Yaskawa INFORM job: DEMO_ROOF_SIDE_0625_3PAINT_0.JBI

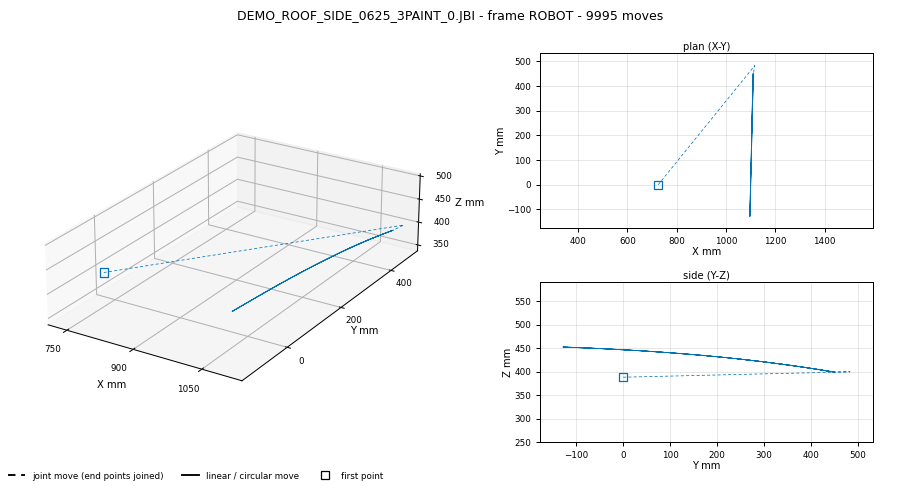
[picture p0: tool path of DEMO_ROOF_SIDE_0625_3PAINT_0.JBI in frame ROBOT, 9995 of 9995 moves have a stored position in this frame; points joined in program order, loops and branches not executed]
/JOB
//NAME DEMO_ROOF_SIDE_0625_3PAINT
//POS
///NPOS 9995,0,0,0,0,0
///TOOL 0
///USER 0
///POSTYPE ROBOT
///RECTAN
///RCONF 1,0,0,0,0,0,0,0,0,0,0,0,0,0,0,0,0,0,0,0,0,0,0,0
C00000=725.000,0.000,388.500,-180.000,-0.000,0.000
///USER 0
///POSTYPE ROBOT
///RECTAN
C00001=1116.924,483.635,399.956,-178.124,16.519,151.125
C00002=1111.077,450.492,399.580,-178.124,16.519,151.125
C00003=1111.072,450.245,399.621,-178.121,16.509,151.122
C00004=1111.067,450.000,399.662,-178.120,16.499,151.119
C00005=1111.061,449.753,399.703,-178.118,16.490,151.116
C00006=1111.056,449.506,399.745,-178.115,16.481,151.114
C00007=1111.050,449.260,399.787,-178.113,16.472,151.111
C00008=1111.045,449.013,399.827,-178.111,16.462,151.108
C00009=1111.039,448.767,399.869,-178.109,16.453,151.105
C00010=1111.034,448.521,399.910,-178.107,16.443,151.102
C00011=1111.028,448.275,399.951,-178.105,16.434,151.099
C00012=1111.023,448.027,399.993,-178.103,16.424,151.096
C00013=1111.017,447.781,400.034,-178.102,16.415,151.094
C00014=1111.012,447.534,400.075,-178.100,16.405,151.091
C00015=1111.007,447.289,400.116,-178.099,16.395,151.088
C00016=1111.002,447.042,400.157,-178.098,16.386,151.085
C00017=1110.996,446.796,400.199,-178.096,16.376,151.082
C00018=1110.991,446.548,400.240,-178.095,16.367,151.080
C00019=1110.985,446.302,400.281,-178.093,16.357,151.077
C00020=1110.980,446.056,400.322,-178.092,16.348,151.074
C00021=1110.975,445.810,400.364,-178.092,16.338,151.072
C00022=1110.969,445.563,400.405,-178.091,16.328,151.069
C00023=1110.963,445.317,400.446,-178.090,16.318,151.066
C00024=1110.957,445.070,400.487,-178.089,16.309,151.064
C00025=1110.952,444.824,400.527,-178.089,16.299,151.061
C00026=1110.947,444.577,400.569,-178.088,16.290,151.058
C00027=1110.941,444.330,400.610,-178.088,16.280,151.056
C00028=1110.935,444.084,400.651,-178.088,16.270,151.053
C00029=1110.930,443.838,400.692,-178.088,16.260,151.051
C00030=1110.925,443.591,400.733,-178.087,16.251,151.048
C00031=1110.919,443.345,400.774,-178.087,16.241,151.046
C00032=1110.915,443.099,400.815,-178.088,16.231,151.043
C00033=1110.909,442.852,400.856,-178.088,16.221,151.041
C00034=1110.903,442.605,400.897,-178.088,16.212,151.038
C00035=1110.898,442.359,400.938,-178.089,16.202,151.036
C00036=1110.892,442.113,400.978,-178.088,16.192,151.033
C00037=1110.887,441.866,401.019,-178.089,16.182,151.031
C00038=1110.881,441.620,401.060,-178.089,16.173,151.028
C00039=1110.876,441.373,401.101,-178.089,16.164,151.026
C00040=1110.870,441.127,401.142,-178.090,16.154,151.024
C00041=1110.864,440.880,401.182,-178.090,16.145,151.021
C00042=1110.859,440.634,401.223,-178.090,16.136,151.019
C00043=1110.853,440.387,401.264,-178.091,16.126,151.017
C00044=1110.848,440.141,401.305,-178.092,16.117,151.014
C00045=1110.843,439.894,401.345,-178.092,16.107,151.012
C00046=1110.837,439.648,401.386,-178.093,16.098,151.010
C00047=1110.831,439.401,401.427,-178.093,16.089,151.007
C00048=1110.826,439.155,401.467,-178.093,16.080,151.005
C00049=1110.820,438.908,401.507,-178.094,16.071,151.003
C00050=1110.814,438.661,401.548,-178.095,16.061,151.001
C00051=1110.809,438.428,401.587,-178.095,16.052,150.998
C00052=1110.804,438.194,401.625,-178.095,16.044,150.996
C00053=1110.799,437.961,401.663,-178.096,16.036,150.994
C00054=1110.794,437.728,401.702,-178.096,16.027,150.992
C00055=1110.788,437.494,401.740,-178.097,16.019,150.990
C00056=1110.783,437.261,401.779,-178.098,16.010,150.988
C00057=1110.778,437.027,401.817,-178.098,16.002,150.986
C00058=1110.773,436.795,401.855,-178.099,15.993,150.984
C00059=1110.767,436.548,401.895,-178.100,15.985,150.982
C00060=1110.761,436.301,401.936,-178.100,15.976,150.980
C00061=1110.756,436.055,401.977,-178.101,15.967,150.978
C00062=1110.751,435.808,402.017,-178.102,15.958,150.976
C00063=1110.745,435.562,402.056,-178.103,15.949,150.973
C00064=1110.740,435.315,402.097,-178.103,15.941,150.971
C00065=1110.734,435.068,402.138,-178.104,15.932,150.969
C00066=1110.729,434.822,402.178,-178.104,15.924,150.967
C00067=1110.723,434.575,402.218,-178.105,15.915,150.965
C00068=1110.718,434.329,402.258,-178.106,15.906,150.963
C00069=1110.712,434.082,402.299,-178.107,15.898,150.961
C00070=1110.707,433.836,402.339,-178.108,15.889,150.959
C00071=1110.701,433.589,402.379,-178.109,15.881,150.957
C00072=1110.696,433.343,402.419,-178.110,15.872,150.955
C00073=1110.690,433.096,402.460,-178.111,15.864,150.953
C00074=1110.684,432.849,402.499,-178.111,15.856,150.951
C00075=1110.679,432.602,402.540,-178.112,15.847,150.949
C00076=1110.674,432.356,402.580,-178.113,15.839,150.947
C00077=1110.668,432.109,402.619,-178.114,15.831,150.945
C00078=1110.662,431.862,402.660,-178.115,15.823,150.943
C00079=1110.657,431.616,402.699,-178.116,15.815,150.942
C00080=1110.651,431.369,402.740,-178.117,15.807,150.940
C00081=1110.646,431.123,402.780,-178.118,15.798,150.938
C00082=1110.640,430.876,402.820,-178.119,15.790,150.936
C00083=1110.635,430.630,402.860,-178.120,15.782,150.934
C00084=1110.629,430.383,402.900,-178.121,15.774,150.932
C00085=1110.623,430.136,402.940,-178.122,15.766,150.930
C00086=1110.618,429.889,402.979,-178.123,15.758,150.928
C00087=1110.612,429.642,403.020,-178.124,15.750,150.927
C00088=1110.607,429.396,403.059,-178.125,15.742,150.925
C00089=1110.602,429.149,403.099,-178.126,15.734,150.923
C00090=1110.596,428.903,403.139,-178.127,15.726,150.921
C00091=1110.590,428.655,403.179,-178.128,15.719,150.919
C00092=1110.585,428.410,403.219,-178.130,15.711,150.918
C00093=1110.579,428.162,403.258,-178.131,15.703,150.916
C00094=1110.574,427.916,403.298,-178.132,15.695,150.914
C00095=1110.567,427.669,403.338,-178.133,15.687,150.912
C00096=1110.563,427.422,403.378,-178.134,15.680,150.911
C00097=1110.557,427.175,403.417,-178.135,15.672,150.909
C00098=1110.551,426.929,403.456,-178.136,15.665,150.907
C00099=1110.546,426.682,403.497,-178.138,15.657,150.906
C00100=1110.540,426.436,403.536,-178.139,15.649,150.904
C00101=1110.534,426.188,403.575,-178.140,15.642,150.902
C00102=1110.529,425.942,403.615,-178.141,15.635,150.901
C00103=1110.523,425.696,403.655,-178.142,15.627,150.899
C00104=1110.518,425.448,403.695,-178.144,15.620,150.897
C00105=1110.513,425.202,403.734,-178.145,15.612,150.896
C00106=1110.507,424.955,403.773,-178.146,15.604,150.894
C00107=1110.502,424.737,403.809,-178.148,15.598,150.893
C00108=1110.497,424.520,403.843,-178.149,15.591,150.891
C00109=1110.492,424.301,403.878,-178.150,15.585,150.890
C00110=1110.487,424.083,403.913,-178.151,15.579,150.888
C00111=1110.483,423.866,403.948,-178.152,15.572,150.887
C00112=1110.477,423.649,403.982,-178.153,15.566,150.885
C00113=1110.472,423.430,404.017,-178.154,15.560,150.884
C00114=1110.468,423.213,404.052,-178.155,15.553,150.883
C00115=1110.462,422.966,404.091,-178.157,15.546,150.881
C00116=1110.456,422.719,404.130,-178.158,15.538,150.880
C00117=1110.451,422.472,404.170,-178.160,15.531,150.878
C00118=1110.446,422.226,404.209,-178.161,15.524,150.877
C00119=1110.440,421.979,404.248,-178.163,15.517,150.875
C00120=1110.434,421.732,404.288,-178.164,15.510,150.874
C00121=1110.429,421.486,404.327,-178.165,15.503,150.872
C00122=1110.422,421.238,404.366,-178.167,15.496,150.871
C00123=1110.417,420.992,404.405,-178.169,15.489,150.869
C00124=1110.412,420.745,404.444,-178.170,15.483,150.868
C00125=1110.407,420.497,404.484,-178.171,15.475,150.866
C00126=1110.401,420.251,404.523,-178.173,15.468,150.865
C00127=1110.395,420.004,404.562,-178.174,15.462,150.863
C00128=1110.389,419.757,404.601,-178.176,15.455,150.862
C00129=1110.384,419.511,404.640,-178.177,15.448,150.860
C00130=1110.378,419.263,404.679,-178.179,15.441,150.859
C00131=1110.373,419.017,404.718,-178.181,15.434,150.858
C00132=1110.367,418.770,404.757,-178.182,15.428,150.856
C00133=1110.361,418.523,404.797,-178.184,15.421,150.855
C00134=1110.356,418.276,404.835,-178.185,15.415,150.854
C00135=1110.351,418.030,404.874,-178.187,15.408,150.852
C00136=1110.345,417.783,404.913,-178.188,15.401,150.851
C00137=1110.339,417.536,404.952,-178.190,15.394,150.850
C00138=1110.334,417.289,404.991,-178.191,15.388,150.848
C00139=1110.328,417.042,405.030,-178.193,15.381,150.847
C00140=1110.323,416.795,405.069,-178.194,15.375,150.845
C00141=1110.317,416.549,405.108,-178.196,15.368,150.844
C00142=1110.311,416.301,405.146,-178.197,15.362,150.843
C00143=1110.306,416.054,405.186,-178.199,15.355,150.842
C00144=1110.301,415.807,405.224,-178.201,15.349,150.840
C00145=1110.295,415.560,405.263,-178.203,15.342,150.839
C00146=1110.288,415.314,405.302,-178.204,15.336,150.838
C00147=1110.283,415.067,405.340,-178.206,15.330,150.836
C00148=1110.277,414.820,405.380,-178.208,15.323,150.835
C00149=1110.272,414.573,405.418,-178.210,15.317,150.834
C00150=1110.267,414.326,405.456,-178.211,15.311,150.833
C00151=1110.261,414.079,405.495,-178.213,15.305,150.832
C00152=1110.255,413.832,405.533,-178.215,15.298,150.830
C00153=1110.249,413.585,405.573,-178.216,15.292,150.829
C00154=1110.244,413.338,405.611,-178.218,15.286,150.828
C00155=1110.238,413.091,405.650,-178.220,15.280,150.827
C00156=1110.232,412.844,405.688,-178.222,15.274,150.826
C00157=1110.227,412.597,405.726,-178.224,15.267,150.824
C00158=1110.222,412.351,405.765,-178.225,15.261,150.823
C00159=1110.216,412.103,405.804,-178.227,15.255,150.822
C00160=1110.211,411.856,405.843,-178.229,15.249,150.821
C00161=1110.205,411.609,405.880,-178.231,15.243,150.820
C00162=1110.199,411.363,405.919,-178.232,15.237,150.818
C00163=1110.194,411.151,405.952,-178.234,15.232,150.818
C00164=1110.190,410.939,405.985,-178.235,15.227,150.817
C00165=1110.185,410.729,406.018,-178.237,15.222,150.816
C00166=1110.180,410.517,406.051,-178.238,15.217,150.815
C00167=1110.176,410.305,406.083,-178.240,15.211,150.814
C00168=1110.171,410.094,406.117,-178.241,15.207,150.813
C00169=1110.166,409.883,406.149,-178.243,15.201,150.812
C00170=1110.161,409.671,406.182,-178.244,15.197,150.811
C00171=1110.156,409.424,406.220,-178.247,15.190,150.810
C00172=1110.150,409.177,406.260,-178.248,15.185,150.809
C00173=1110.144,408.931,406.297,-178.250,15.179,150.808
C00174=1110.139,408.683,406.336,-178.252,15.173,150.806
C00175=1110.134,408.436,406.374,-178.253,15.168,150.805
C00176=1110.128,408.190,406.412,-178.256,15.161,150.804
C00177=1110.123,407.943,406.450,-178.258,15.156,150.803
C00178=1110.116,407.695,406.488,-178.259,15.150,150.802
C00179=1110.111,407.448,406.527,-178.261,15.145,150.801
C00180=1110.105,407.201,406.564,-178.263,15.139,150.800
C00181=1110.100,406.954,406.603,-178.266,15.133,150.799
C00182=1110.095,406.707,406.641,-178.267,15.127,150.798
C00183=1110.089,406.461,406.679,-178.269,15.122,150.797
C00184=1110.084,406.213,406.717,-178.271,15.116,150.796
C00185=1110.077,405.966,406.755,-178.273,15.111,150.795
C00186=1110.072,405.719,406.794,-178.275,15.105,150.794
C00187=1110.066,405.472,406.831,-178.277,15.100,150.793
C00188=1110.061,405.225,406.870,-178.279,15.095,150.792
C00189=1110.055,404.978,406.907,-178.281,15.089,150.791
C00190=1110.049,404.731,406.944,-178.283,15.084,150.791
C00191=1110.044,404.484,406.983,-178.285,15.078,150.790
C00192=1110.038,404.237,407.021,-178.287,15.073,150.789
C00193=1110.033,403.989,407.059,-178.289,15.067,150.788
C00194=1110.027,403.743,407.097,-178.291,15.062,150.787
C00195=1110.021,403.496,407.135,-178.293,15.057,150.786
C00196=1110.016,403.248,407.172,-178.295,15.051,150.785
C00197=1110.010,403.002,407.210,-178.297,15.046,150.784
C00198=1110.004,402.755,407.248,-178.299,15.041,150.783
C00199=1109.999,402.508,407.286,-178.301,15.035,150.782
C00200=1109.993,402.260,407.323,-178.303,15.030,150.781
C00201=1109.987,402.014,407.361,-178.305,15.025,150.781
C00202=1109.982,401.767,407.399,-178.307,15.020,150.780
C00203=1109.977,401.519,407.437,-178.309,15.014,150.779
C00204=1109.971,401.273,407.474,-178.312,15.009,150.778
C00205=1109.966,401.025,407.513,-178.313,15.004,150.777
C00206=1109.960,400.778,407.550,-178.316,14.999,150.776
C00207=1109.954,400.531,407.587,-178.317,14.995,150.775
C00208=1109.949,400.284,407.625,-178.319,14.989,150.775
C00209=1109.943,400.037,407.663,-178.321,14.984,150.774
C00210=1109.937,399.790,407.701,-178.324,14.979,150.773
C00211=1109.932,399.543,407.738,-178.326,14.974,150.772
C00212=1109.926,399.296,407.775,-178.328,14.969,150.771
C00213=1109.921,399.048,407.813,-178.330,14.964,150.771
C00214=1109.915,398.801,407.851,-178.332,14.959,150.770
C00215=1109.909,398.554,407.888,-178.335,14.954,150.769
C00216=1109.904,398.308,407.926,-178.337,14.949,150.768
C00217=1109.898,398.060,407.963,-178.339,14.945,150.767
C00218=1109.892,397.813,408.000,-178.341,14.940,150.767
C00219=1109.888,397.601,408.033,-178.343,14.936,150.766
C00220=1109.883,397.390,408.065,-178.345,14.931,150.765
C00221=1109.878,397.178,408.096,-178.347,14.927,150.765
C00222=1109.873,396.966,408.129,-178.349,14.923,150.764
C00223=1109.868,396.755,408.161,-178.350,14.919,150.763
C00224=1109.863,396.543,408.192,-178.352,14.915,150.763
C00225=1109.858,396.331,408.225,-178.354,14.911,150.762
C00226=1109.854,396.119,408.257,-178.356,14.907,150.762
C00227=1109.848,395.872,408.294,-178.358,14.902,150.761
C00228=1109.842,395.625,408.331,-178.360,14.897,150.760
C00229=1109.837,395.378,408.368,-178.363,14.892,150.760
C00230=1109.831,395.132,408.406,-178.365,14.887,150.759
C00231=1109.826,394.884,408.443,-178.367,14.883,150.758
C00232=1109.820,394.637,408.480,-178.369,14.878,150.757
C00233=1109.815,394.389,408.517,-178.372,14.874,150.757
C00234=1109.809,394.143,408.555,-178.374,14.869,150.756
C00235=1109.803,393.895,408.592,-178.376,14.865,150.755
C00236=1109.797,393.648,408.629,-178.379,14.860,150.755
C00237=1109.792,393.401,408.666,-178.381,14.855,150.754
C00238=1109.787,393.155,408.703,-178.383,14.850,150.753
C00239=1109.781,392.907,408.740,-178.385,14.847,150.753
C00240=1109.775,392.660,408.777,-178.387,14.842,150.752
C00241=1109.770,392.413,408.814,-178.390,14.837,150.752
C00242=1109.764,392.165,408.851,-178.393,14.832,150.751
C00243=1109.758,391.918,408.888,-178.394,14.828,150.750
C00244=1109.752,391.671,408.926,-178.397,14.824,150.750
C00245=1109.746,391.424,408.963,-178.400,14.819,150.749
C00246=1109.741,391.177,408.999,-178.401,14.815,150.749
C00247=1109.736,390.930,409.036,-178.404,14.811,150.748
C00248=1109.729,390.683,409.073,-178.407,14.806,150.748
C00249=1109.724,390.436,409.110,-178.410,14.802,150.747
C00250=1109.718,390.188,409.147,-178.411,14.798,150.746
C00251=1109.713,389.942,409.184,-178.414,14.793,150.746
C00252=1109.707,389.694,409.220,-178.417,14.788,150.745
C00253=1109.701,389.447,409.257,-178.419,14.785,150.745
C00254=1109.696,389.200,409.294,-178.421,14.780,150.744
C00255=1109.690,388.952,409.331,-178.424,14.776,150.744
C00256=1109.684,388.706,409.367,-178.426,14.772,150.743
C00257=1109.679,388.459,409.404,-178.429,14.767,150.743
C00258=1109.673,388.211,409.441,-178.432,14.763,150.742
C00259=1109.667,387.964,409.478,-178.433,14.759,150.741
C00260=1109.662,387.718,409.514,-178.436,14.755,150.741
C00261=1109.656,387.470,409.551,-178.438,14.751,150.740
C00262=1109.650,387.223,409.588,-178.441,14.747,150.740
C00263=1109.645,386.976,409.624,-178.444,14.742,150.739
C00264=1109.640,386.729,409.661,-178.446,14.738,150.739
C00265=1109.633,386.481,409.697,-178.448,14.734,150.738
C00266=1109.628,386.234,409.734,-178.451,14.729,150.738
C00267=1109.623,385.987,409.771,-178.453,14.726,150.738
C00268=1109.617,385.740,409.807,-178.456,14.721,150.737
C00269=1109.611,385.492,409.844,-178.458,14.718,150.737
C00270=1109.606,385.246,409.880,-178.461,14.713,150.736
C00271=1109.600,384.999,409.917,-178.464,14.709,150.736
C00272=1109.594,384.751,409.953,-178.466,14.706,150.735
C00273=1109.589,384.504,409.989,-178.469,14.701,150.735
C00274=1109.583,384.257,410.026,-178.471,14.697,150.734
C00275=1109.573,383.845,410.087,-178.476,14.691,150.734
C00276=1109.564,383.434,410.147,-178.479,14.684,150.733
C00277=1109.555,383.023,410.208,-178.484,14.677,150.732
C00278=1109.546,382.612,410.268,-178.488,14.671,150.732
C00279=1109.540,382.364,410.305,-178.491,14.667,150.731
C00280=1109.534,382.117,410.341,-178.493,14.663,150.731
C00281=1109.529,381.870,410.377,-178.496,14.660,150.730
C00282=1109.523,381.622,410.413,-178.498,14.656,150.730
C00283=1109.517,381.375,410.450,-178.501,14.652,150.730
C00284=1109.512,381.128,410.486,-178.504,14.649,150.729
C00285=1109.506,380.881,410.522,-178.507,14.644,150.729
C00286=1109.500,380.633,410.558,-178.509,14.641,150.728
C00287=1109.495,380.386,410.595,-178.512,14.637,150.728
C00288=1109.489,380.139,410.630,-178.514,14.633,150.728
C00289=1109.483,379.891,410.667,-178.517,14.629,150.728
C00290=1109.478,379.644,410.703,-178.520,14.626,150.727
C00291=1109.472,379.397,410.739,-178.523,14.622,150.727
C00292=1109.467,379.150,410.775,-178.525,14.618,150.726
C00293=1109.461,378.902,410.811,-178.528,14.614,150.726
C00294=1109.455,378.656,410.847,-178.530,14.611,150.726
C00295=1109.450,378.408,410.883,-178.533,14.608,150.726
C00296=1109.444,378.160,410.919,-178.536,14.604,150.725
C00297=1109.438,377.914,410.955,-178.538,14.600,150.725
C00298=1109.433,377.666,410.991,-178.542,14.596,150.725
C00299=1109.427,377.419,411.027,-178.544,14.593,150.724
C00300=1109.421,377.171,411.063,-178.547,14.589,150.724
C00301=1109.416,376.925,411.099,-178.549,14.585,150.724
C00302=1109.410,376.677,411.135,-178.552,14.582,150.723
C00303=1109.405,376.430,411.170,-178.555,14.578,150.723
C00304=1109.399,376.182,411.206,-178.557,14.575,150.723
C00305=1109.393,375.936,411.242,-178.561,14.571,150.723
C00306=1109.388,375.688,411.278,-178.563,14.568,150.722
C00307=1109.382,375.441,411.314,-178.566,14.564,150.722
C00308=1109.376,375.194,411.350,-178.569,14.561,150.722
C00309=1109.371,374.947,411.385,-178.571,14.557,150.722
C00310=1109.366,374.699,411.421,-178.574,14.554,150.721
C00311=1109.360,374.452,411.457,-178.577,14.550,150.721
C00312=1109.354,374.205,411.493,-178.580,14.547,150.721
C00313=1109.348,373.957,411.529,-178.583,14.543,150.721
C00314=1109.342,373.710,411.564,-178.585,14.540,150.720
C00315=1109.336,373.462,411.600,-178.588,14.537,150.720
C00316=1109.331,373.215,411.635,-178.591,14.533,150.720
C00317=1109.325,372.968,411.671,-178.594,14.530,150.720
C00318=1109.319,372.721,411.706,-178.596,14.527,150.719
C00319=1109.314,372.473,411.743,-178.599,14.524,150.719
C00320=1109.309,372.226,411.778,-178.602,14.520,150.719
C00321=1109.303,371.978,411.814,-178.605,14.517,150.719
C00322=1109.297,371.731,411.849,-178.608,14.514,150.719
C00323=1109.291,371.483,411.885,-178.611,14.510,150.719
C00324=1109.286,371.236,411.920,-178.614,14.507,150.718
C00325=1109.280,370.989,411.956,-178.616,14.504,150.718
C00326=1109.274,370.742,411.991,-178.620,14.500,150.718
C00327=1109.266,370.357,412.046,-178.624,14.495,150.718
C00328=1109.256,369.972,412.101,-178.628,14.491,150.718
C00329=1109.248,369.587,412.156,-178.633,14.485,150.717
C00330=1109.240,369.202,412.211,-178.637,14.481,150.717
C00331=1109.233,368.955,412.247,-178.640,14.478,150.717
C00332=1109.228,368.708,412.282,-178.643,14.474,150.717
C00333=1109.222,368.459,412.317,-178.646,14.471,150.717
C00334=1109.217,368.212,412.352,-178.649,14.468,150.717
C00335=1109.211,367.966,412.388,-178.651,14.465,150.716
C00336=1109.206,367.717,412.423,-178.655,14.461,150.716
C00337=1109.200,367.471,412.458,-178.658,14.459,150.716
C00338=1109.194,367.224,412.493,-178.661,14.456,150.716
C00339=1109.188,366.975,412.528,-178.663,14.453,150.716
C00340=1109.183,366.728,412.563,-178.667,14.449,150.716
C00341=1109.177,366.481,412.599,-178.669,14.446,150.716
C00342=1109.172,366.233,412.634,-178.672,14.443,150.716
C00343=1109.166,365.986,412.669,-178.675,14.441,150.716
C00344=1109.160,365.738,412.705,-178.678,14.438,150.716
C00345=1109.155,365.491,412.739,-178.681,14.434,150.715
C00346=1109.149,365.244,412.774,-178.684,14.431,150.715
C00347=1109.143,364.996,412.809,-178.687,14.428,150.715
C00348=1109.138,364.749,412.845,-178.690,14.426,150.715
C00349=1109.132,364.501,412.880,-178.693,14.423,150.715
C00350=1109.126,364.254,412.914,-178.696,14.419,150.715
C00351=1109.121,364.006,412.949,-178.699,14.416,150.715
C00352=1109.115,363.759,412.985,-178.702,14.414,150.715
C00353=1109.110,363.511,413.019,-178.705,14.411,150.715
C00354=1109.104,363.264,413.054,-178.708,14.408,150.715
C00355=1109.098,363.016,413.089,-178.711,14.405,150.715
C00356=1109.092,362.769,413.125,-178.714,14.402,150.715
C00357=1109.087,362.522,413.159,-178.717,14.399,150.715
C00358=1109.081,362.274,413.193,-178.720,14.396,150.715
C00359=1109.075,362.027,413.229,-178.723,14.393,150.715
C00360=1109.070,361.779,413.263,-178.726,14.391,150.715
C00361=1109.064,361.532,413.298,-178.729,14.388,150.715
C00362=1109.058,361.284,413.333,-178.732,14.385,150.715
C00363=1109.053,361.037,413.367,-178.736,14.382,150.715
C00364=1109.047,360.789,413.402,-178.739,14.379,150.715
C00365=1109.041,360.541,413.438,-178.741,14.376,150.715
C00366=1109.036,360.294,413.472,-178.745,14.374,150.715
C00367=1109.030,360.047,413.507,-178.747,14.371,150.715
C00368=1109.024,359.800,413.541,-178.751,14.369,150.715
C00369=1109.019,359.552,413.576,-178.753,14.366,150.715
C00370=1109.013,359.304,413.610,-178.757,14.363,150.715
C00371=1109.008,359.057,413.645,-178.759,14.361,150.715
C00372=1109.002,358.809,413.680,-178.763,14.358,150.715
C00373=1108.996,358.562,413.715,-178.767,14.355,150.715
C00374=1108.991,358.314,413.749,-178.769,14.352,150.715
C00375=1108.985,358.067,413.784,-178.773,14.350,150.715
C00376=1108.980,357.819,413.818,-178.775,14.347,150.715
C00377=1108.973,357.571,413.853,-178.779,14.344,150.715
C00378=1108.968,357.324,413.887,-178.782,14.342,150.715
C00379=1108.959,356.954,413.939,-178.786,14.338,150.715
C00380=1108.950,356.584,413.990,-178.791,14.334,150.715
C00381=1108.942,356.214,414.042,-178.796,14.330,150.715
C00382=1108.934,355.844,414.093,-178.800,14.326,150.715
C00383=1108.928,355.596,414.128,-178.803,14.324,150.716
C00384=1108.922,355.348,414.162,-178.806,14.322,150.716
C00385=1108.917,355.101,414.196,-178.810,14.319,150.716
C00386=1108.911,354.854,414.230,-178.813,14.317,150.716
C00387=1108.906,354.606,414.265,-178.816,14.314,150.716
C00388=1108.900,354.358,414.299,-178.819,14.311,150.716
C00389=1108.894,354.110,414.334,-178.822,14.309,150.716
C00390=1108.889,353.863,414.368,-178.825,14.306,150.716
C00391=1108.883,353.616,414.402,-178.828,14.304,150.716
C00392=1108.878,353.368,414.436,-178.832,14.302,150.716
C00393=1108.872,353.120,414.470,-178.835,14.299,150.716
C00394=1108.866,352.873,414.504,-178.838,14.297,150.717
C00395=1108.860,352.625,414.539,-178.841,14.294,150.717
C00396=1108.855,352.377,414.573,-178.844,14.292,150.717
C00397=1108.849,352.130,414.607,-178.848,14.290,150.717
C00398=1108.843,351.882,414.641,-178.851,14.287,150.717
C00399=1108.838,351.635,414.675,-178.854,14.285,150.717
C00400=1108.832,351.387,414.709,-178.857,14.282,150.717
C00401=1108.826,351.140,414.743,-178.861,14.280,150.718
C00402=1108.820,350.892,414.777,-178.864,14.277,150.718
C00403=1108.815,350.644,414.812,-178.867,14.275,150.718
C00404=1108.809,350.397,414.846,-178.870,14.273,150.718
C00405=1108.804,350.149,414.879,-178.874,14.270,150.718
C00406=1108.798,349.901,414.913,-178.877,14.268,150.718
C00407=1108.792,349.654,414.947,-178.880,14.266,150.719
C00408=1108.787,349.406,414.981,-178.883,14.263,150.719
C00409=1108.781,349.159,415.015,-178.887,14.261,150.719
C00410=1108.775,348.911,415.049,-178.890,14.259,150.719
C00411=1108.770,348.664,415.083,-178.893,14.256,150.719
C00412=1108.763,348.416,415.117,-178.897,14.254,150.719
C00413=1108.758,348.168,415.150,-178.900,14.252,150.720
C00414=1108.753,347.920,415.185,-178.903,14.249,150.720
C00415=1108.747,347.673,415.219,-178.906,14.248,150.720
C00416=1108.741,347.425,415.252,-178.909,14.246,150.720
C00417=1108.735,347.178,415.287,-178.912,14.243,150.720
C00418=1108.730,346.930,415.320,-178.916,14.241,150.720
C00419=1108.724,346.682,415.354,-178.919,14.239,150.721
C00420=1108.718,346.434,415.387,-178.923,14.237,150.721
C00421=1108.713,346.187,415.421,-178.926,14.234,150.721
C00422=1108.707,345.939,415.455,-178.929,14.232,150.721
C00423=1108.701,345.691,415.488,-178.932,14.230,150.721
C00424=1108.696,345.444,415.523,-178.936,14.228,150.722
C00425=1108.691,345.196,415.556,-178.939,14.226,150.722
C00426=1108.685,344.949,415.590,-178.942,14.224,150.722
C00427=1108.679,344.701,415.623,-178.946,14.222,150.722
C00428=1108.673,344.453,415.656,-178.949,14.220,150.723
C00429=1108.667,344.206,415.690,-178.952,14.217,150.723
C00430=1108.662,343.958,415.723,-178.956,14.215,150.723
C00431=1108.654,343.590,415.773,-178.961,14.212,150.724
C00432=1108.645,343.223,415.823,-178.965,14.209,150.724
C00433=1108.636,342.854,415.873,-178.971,14.206,150.724
C00434=1108.628,342.486,415.923,-178.976,14.203,150.725
C00435=1108.622,342.238,415.956,-178.978,14.201,150.725
C00436=1108.616,341.991,415.990,-178.982,14.199,150.725
C00437=1108.611,341.743,416.023,-178.985,14.197,150.725
C00438=1108.605,341.495,416.056,-178.989,14.195,150.726
C00439=1108.600,341.247,416.090,-178.992,14.193,150.726
C00440=1108.594,340.999,416.123,-178.996,14.191,150.726
C00441=1108.589,340.751,416.156,-178.999,14.189,150.727
C00442=1108.583,340.505,416.190,-179.002,14.187,150.727
C00443=1108.577,340.257,416.223,-179.006,14.185,150.727
C00444=1108.571,340.009,416.256,-179.009,14.183,150.727
C00445=1108.566,339.761,416.290,-179.012,14.181,150.728
C00446=1108.560,339.513,416.323,-179.015,14.179,150.728
C00447=1108.555,339.265,416.356,-179.019,14.177,150.728
C00448=1108.549,339.017,416.390,-179.022,14.175,150.728
C00449=1108.543,338.770,416.422,-179.026,14.173,150.729
C00450=1108.537,338.522,416.456,-179.029,14.171,150.729
C00451=1108.532,338.274,416.489,-179.032,14.170,150.729
C00452=1108.527,338.027,416.522,-179.036,14.168,150.730
C00453=1108.521,337.779,416.555,-179.040,14.166,150.730
C00454=1108.515,337.531,416.588,-179.043,14.164,150.730
C00455=1108.509,337.283,416.621,-179.046,14.163,150.731
C00456=1108.503,337.036,416.654,-179.049,14.161,150.731
C00457=1108.498,336.788,416.687,-179.053,14.159,150.731
C00458=1108.492,336.540,416.721,-179.057,14.157,150.732
C00459=1108.486,336.292,416.754,-179.060,14.155,150.732
C00460=1108.481,336.045,416.786,-179.063,14.153,150.732
C00461=1108.476,335.797,416.819,-179.067,14.151,150.733
C00462=1108.469,335.549,416.852,-179.071,14.150,150.733
C00463=1108.464,335.301,416.885,-179.073,14.148,150.733
C00464=1108.458,335.053,416.919,-179.077,14.146,150.734
C00465=1108.452,334.806,416.951,-179.080,14.144,150.734
C00466=1108.447,334.558,416.984,-179.084,14.142,150.734
C00467=1108.441,334.310,417.016,-179.087,14.141,150.735
C00468=1108.435,334.062,417.050,-179.091,14.139,150.735
C00469=1108.430,333.814,417.083,-179.094,14.137,150.736
C00470=1108.423,333.567,417.116,-179.098,14.135,150.736
C00471=1108.419,333.319,417.148,-179.101,14.134,150.736
C00472=1108.413,333.071,417.181,-179.105,14.132,150.737
C00473=1108.407,332.824,417.214,-179.108,14.130,150.737
C00474=1108.402,332.575,417.247,-179.111,14.129,150.737
C00475=1108.395,332.327,417.279,-179.115,14.127,150.738
C00476=1108.391,332.080,417.312,-179.119,14.126,150.738
C00477=1108.385,331.832,417.344,-179.122,14.124,150.738
C00478=1108.378,331.584,417.377,-179.125,14.122,150.739
C00479=1108.373,331.337,417.410,-179.129,14.120,150.739
C00480=1108.367,331.088,417.442,-179.132,14.119,150.740
C00481=1108.361,330.841,417.475,-179.136,14.118,150.740
C00482=1108.356,330.593,417.507,-179.139,14.116,150.740
C00483=1108.347,330.219,417.558,-179.144,14.114,150.741
C00484=1108.338,329.845,417.606,-179.150,14.111,150.742
C00485=1108.329,329.471,417.656,-179.155,14.109,150.742
C00486=1108.321,329.097,417.705,-179.161,14.106,150.743
C00487=1108.315,328.849,417.737,-179.164,14.105,150.743
C00488=1108.309,328.601,417.769,-179.168,14.104,150.744
C00489=1108.304,328.353,417.802,-179.171,14.102,150.744
C00490=1108.298,328.105,417.834,-179.174,14.101,150.745
C00491=1108.292,327.857,417.867,-179.178,14.099,150.745
C00492=1108.286,327.609,417.899,-179.182,14.097,150.746
C00493=1108.281,327.362,417.931,-179.185,14.096,150.746
C00494=1108.275,327.114,417.964,-179.189,14.094,150.746
C00495=1108.269,326.865,417.996,-179.192,14.093,150.747
C00496=1108.264,326.618,418.029,-179.196,14.092,150.747
C00497=1108.258,326.370,418.061,-179.200,14.090,150.748
C00498=1108.252,326.122,418.093,-179.202,14.089,150.748
C00499=1108.246,325.875,418.125,-179.206,14.087,150.749
C00500=1108.241,325.626,418.158,-179.210,14.085,150.749
C00501=1108.235,325.378,418.190,-179.213,14.084,150.750
C00502=1108.229,325.131,418.222,-179.217,14.083,150.750
C00503=1108.223,324.883,418.254,-179.220,14.082,150.751
C00504=1108.218,324.635,418.287,-179.224,14.080,150.751
C00505=1108.213,324.387,418.318,-179.228,14.078,150.751
C00506=1108.206,324.140,418.351,-179.231,14.077,150.752
C00507=1108.200,323.891,418.383,-179.235,14.075,150.752
C00508=1108.195,323.644,418.415,-179.238,14.074,150.753
C00509=1108.189,323.396,418.447,-179.242,14.073,150.753
C00510=1108.184,323.148,418.479,-179.245,14.072,150.754
C00511=1108.178,322.900,418.512,-179.249,14.070,150.754
C00512=1108.172,322.652,418.544,-179.253,14.068,150.755
C00513=1108.167,322.404,418.575,-179.256,14.067,150.755
C00514=1108.161,322.156,418.607,-179.260,14.066,150.756
C00515=1108.155,321.909,418.639,-179.263,14.065,150.756
C00516=1108.150,321.660,418.672,-179.267,14.063,150.757
C00517=1108.145,321.413,418.703,-179.270,14.062,150.757
C00518=1108.139,321.164,418.735,-179.274,14.060,150.758
C00519=1108.133,320.917,418.767,-179.278,14.059,150.758
C00520=1108.127,320.669,418.799,-179.281,14.058,150.759
C00521=1108.122,320.421,418.831,-179.285,14.056,150.759
C00522=1108.116,320.173,418.863,-179.288,14.055,150.759
C00523=1108.111,319.925,418.894,-179.292,14.054,150.760
C00524=1108.105,319.677,418.926,-179.295,14.053,150.760
C00525=1108.099,319.430,418.958,-179.299,14.051,150.761
C00526=1108.093,319.182,418.990,-179.302,14.050,150.762
C00527=1108.088,318.934,419.022,-179.306,14.049,150.762
C00528=1108.082,318.686,419.054,-179.309,14.048,150.763
C00529=1108.077,318.438,419.086,-179.313,14.046,150.763
C00530=1108.071,318.190,419.118,-179.316,14.045,150.764
C00531=1108.066,317.942,419.150,-179.320,14.043,150.764
C00532=1108.060,317.694,419.182,-179.324,14.042,150.765
C00533=1108.055,317.446,419.213,-179.328,14.041,150.765
C00534=1108.049,317.198,419.245,-179.332,14.040,150.766
C00535=1108.040,316.817,419.294,-179.337,14.038,150.766
C00536=1108.031,316.436,419.342,-179.342,14.036,150.767
C00537=1108.023,316.055,419.390,-179.348,14.034,150.768
C00538=1108.014,315.673,419.439,-179.353,14.032,150.769
C00539=1108.009,315.426,419.471,-179.357,14.031,150.769
C00540=1108.003,315.178,419.503,-179.360,14.030,150.770
C00541=1107.997,314.930,419.534,-179.364,14.028,150.770
C00542=1107.992,314.681,419.566,-179.368,14.028,150.771
C00543=1107.985,314.434,419.597,-179.372,14.026,150.772
C00544=1107.980,314.187,419.628,-179.375,14.025,150.772
C00545=1107.974,313.938,419.660,-179.378,14.025,150.773
C00546=1107.968,313.690,419.691,-179.383,14.023,150.773
C00547=1107.962,313.442,419.723,-179.386,14.022,150.774
C00548=1107.957,313.194,419.754,-179.390,14.021,150.774
C00549=1107.951,312.946,419.786,-179.393,14.020,150.775
C00550=1107.945,312.699,419.817,-179.397,14.019,150.776
C00551=1107.939,312.450,419.848,-179.401,14.018,150.776
C00552=1107.934,312.202,419.880,-179.405,14.017,150.777
C00553=1107.928,311.955,419.910,-179.408,14.016,150.777
C00554=1107.922,311.706,419.942,-179.412,14.014,150.778
C00555=1107.917,311.459,419.974,-179.416,14.014,150.779
C00556=1107.911,311.211,420.004,-179.419,14.013,150.779
C00557=1107.905,310.963,420.036,-179.423,14.012,150.780
C00558=1107.900,310.715,420.067,-179.427,14.011,150.780
C00559=1107.893,310.467,420.098,-179.430,14.009,150.781
C00560=1107.888,310.219,420.129,-179.434,14.009,150.782
C00561=1107.882,309.971,420.160,-179.438,14.007,150.782
C00562=1107.876,309.723,420.192,-179.441,14.007,150.783
C00563=1107.871,309.475,420.223,-179.446,14.005,150.783
C00564=1107.865,309.227,420.254,-179.449,14.004,150.784
C00565=1107.859,308.978,420.285,-179.452,14.004,150.785
C00566=1107.853,308.731,420.316,-179.456,14.003,150.785
C00567=1107.848,308.483,420.347,-179.460,14.002,150.786
C00568=1107.842,308.236,420.378,-179.464,14.000,150.786
C00569=1107.836,307.987,420.409,-179.467,14.000,150.787
C00570=1107.831,307.739,420.440,-179.472,13.999,150.788
C00571=1107.825,307.492,420.472,-179.475,13.998,150.788
C00572=1107.820,307.243,420.503,-179.478,13.997,150.789
C00573=1107.814,306.995,420.533,-179.483,13.996,150.789
C00574=1107.808,306.748,420.565,-179.486,13.995,150.790
C00575=1107.803,306.500,420.595,-179.490,13.994,150.791
C00576=1107.797,306.251,420.626,-179.493,13.993,150.791
C00577=1107.791,306.003,420.657,-179.498,13.992,150.792
C00578=1107.786,305.756,420.689,-179.501,13.991,150.792
C00579=1107.780,305.508,420.719,-179.504,13.990,150.793
C00580=1107.775,305.260,420.750,-179.509,13.989,150.794
C00581=1107.768,305.011,420.781,-179.512,13.989,150.794
C00582=1107.763,304.763,420.811,-179.516,13.987,150.795
C00583=1107.757,304.516,420.843,-179.519,13.986,150.796
C00584=1107.751,304.268,420.873,-179.523,13.986,150.796
C00585=1107.746,304.020,420.904,-179.527,13.985,150.797
C00586=1107.740,303.772,420.934,-179.531,13.984,150.798
C00587=1107.732,303.394,420.981,-179.536,13.983,150.799
C00588=1107.723,303.014,421.028,-179.543,13.981,150.800
C00589=1107.714,302.636,421.075,-179.548,13.979,150.800
C00590=1107.705,302.257,421.122,-179.554,13.978,150.801
C00591=1107.700,302.009,421.153,-179.557,13.978,150.802
C00592=1107.694,301.762,421.183,-179.561,13.976,150.803
C00593=1107.689,301.513,421.214,-179.565,13.976,150.803
C00594=1107.683,301.266,421.245,-179.568,13.975,150.804
C00595=1107.678,301.018,421.275,-179.573,13.974,150.805
C00596=1107.673,300.770,421.306,-179.576,13.974,150.806
C00597=1107.667,300.521,421.336,-179.580,13.972,150.806
C00598=1107.661,300.273,421.366,-179.584,13.972,150.807
C00599=1107.655,300.025,421.397,-179.587,13.971,150.807
C00600=1107.650,299.777,421.428,-179.591,13.970,150.808
C00601=1107.644,299.529,421.458,-179.595,13.969,150.809
C00602=1107.639,299.281,421.489,-179.598,13.969,150.809
C00603=1107.633,299.033,421.519,-179.603,13.967,150.810
C00604=1107.627,298.785,421.550,-179.606,13.967,150.811
C00605=1107.621,298.537,421.580,-179.610,13.966,150.811
C00606=1107.617,298.289,421.610,-179.614,13.965,150.812
C00607=1107.611,298.041,421.641,-179.617,13.964,150.813
C00608=1107.605,297.793,421.671,-179.621,13.964,150.813
C00609=1107.599,297.545,421.701,-179.625,13.963,150.814
C00610=1107.593,297.297,421.732,-179.629,13.963,150.815
C00611=1107.588,297.049,421.761,-179.632,13.962,150.816
C00612=1107.583,296.801,421.792,-179.637,13.961,150.816
C00613=1107.577,296.553,421.823,-179.640,13.960,150.817
C00614=1107.571,296.305,421.853,-179.644,13.960,150.818
C00615=1107.565,296.056,421.883,-179.648,13.959,150.818
C00616=1107.559,295.808,421.913,-179.652,13.958,150.819
C00617=1107.553,295.560,421.944,-179.655,13.958,150.820
C00618=1107.548,295.312,421.973,-179.660,13.957,150.820
C00619=1107.542,295.064,422.004,-179.663,13.956,150.821
C00620=1107.536,294.816,422.034,-179.667,13.956,150.822
C00621=1107.531,294.568,422.064,-179.670,13.955,150.823
C00622=1107.525,294.320,422.094,-179.675,13.954,150.823
C00623=1107.519,294.072,422.124,-179.678,13.954,150.824
C00624=1107.514,293.824,422.154,-179.682,13.953,150.825
C00625=1107.508,293.576,422.184,-179.686,13.952,150.825
C00626=1107.502,293.327,422.214,-179.690,13.951,150.826
C00627=1107.496,293.080,422.244,-179.693,13.951,150.827
C00628=1107.491,292.831,422.274,-179.698,13.950,150.828
C00629=1107.485,292.583,422.304,-179.701,13.949,150.828
C00630=1107.479,292.335,422.335,-179.705,13.949,150.829
C00631=1107.474,292.087,422.364,-179.709,13.949,150.830
C00632=1107.468,291.839,422.394,-179.713,13.948,150.830
C00633=1107.462,291.591,422.424,-179.716,13.947,150.831
C00634=1107.457,291.342,422.454,-179.720,13.947,150.832
C00635=1107.451,291.094,422.484,-179.724,13.946,150.833
C00636=1107.446,290.846,422.514,-179.728,13.945,150.833
C00637=1107.440,290.598,422.544,-179.732,13.945,150.834
C00638=1107.435,290.350,422.574,-179.735,13.945,150.835
C00639=1107.426,289.985,422.617,-179.741,13.943,150.836
C00640=1107.418,289.621,422.661,-179.747,13.943,150.837
C00641=1107.410,289.256,422.705,-179.753,13.942,150.838
C00642=1107.401,288.891,422.749,-179.758,13.941,150.839
C00643=1107.395,288.643,422.779,-179.762,13.940,150.840
C00644=1107.389,288.395,422.808,-179.766,13.940,150.841
C00645=1107.384,288.147,422.838,-179.769,13.940,150.842
C00646=1107.378,287.899,422.868,-179.773,13.939,150.842
C00647=1107.372,287.651,422.898,-179.778,13.938,150.843
C00648=1107.367,287.403,422.926,-179.781,13.938,150.844
C00649=1107.361,287.155,422.956,-179.785,13.938,150.845
C00650=1107.355,286.907,422.986,-179.789,13.937,150.845
C00651=1107.350,286.658,423.016,-179.792,13.937,150.846
C00652=1107.343,286.410,423.045,-179.797,13.936,150.847
C00653=1107.338,286.162,423.075,-179.800,13.936,150.848
C00654=1107.332,285.913,423.104,-179.804,13.935,150.848
C00655=1107.327,285.665,423.134,-179.808,13.935,150.849
C00656=1107.321,285.418,423.163,-179.812,13.934,150.850
C00657=1107.315,285.170,423.193,-179.816,13.934,150.851
C00658=1107.310,284.921,423.223,-179.820,13.933,150.851
C00659=1107.304,284.673,423.252,-179.823,13.933,150.852
C00660=1107.298,284.425,423.281,-179.827,13.933,150.853
C00661=1107.293,284.176,423.311,-179.832,13.932,150.854
C00662=1107.287,283.929,423.340,-179.835,13.931,150.855
C00663=1107.282,283.680,423.369,-179.839,13.931,150.855
C00664=1107.276,283.432,423.399,-179.843,13.931,150.856
C00665=1107.270,283.184,423.428,-179.847,13.930,150.857
C00666=1107.264,282.935,423.457,-179.851,13.930,150.858
C00667=1107.259,282.688,423.487,-179.854,13.929,150.858
C00668=1107.253,282.440,423.516,-179.858,13.929,150.859
C00669=1107.248,282.191,423.545,-179.862,13.929,150.860
C00670=1107.242,281.943,423.575,-179.866,13.928,150.861
C00671=1107.236,281.695,423.604,-179.870,13.927,150.862
C00672=1107.231,281.447,423.633,-179.874,13.927,150.862
C00673=1107.225,281.199,423.662,-179.878,13.927,150.863
C00674=1107.219,280.950,423.692,-179.881,13.926,150.864
C00675=1107.213,280.702,423.721,-179.885,13.926,150.865
C00676=1107.208,280.454,423.750,-179.890,13.926,150.866
C00677=1107.202,280.206,423.779,-179.893,13.925,150.866
C00678=1107.197,279.957,423.808,-179.897,13.925,150.867
C00679=1107.190,279.709,423.837,-179.901,13.925,150.868
C00680=1107.185,279.461,423.867,-179.904,13.924,150.869
C00681=1107.179,279.213,423.896,-179.909,13.924,150.870
C00682=1107.174,278.965,423.925,-179.913,13.923,150.870
C00683=1107.168,278.716,423.954,-179.916,13.923,150.871
C00684=1107.162,278.468,423.983,-179.920,13.923,150.872
C00685=1107.157,278.220,424.012,-179.924,13.923,150.873
C00686=1107.151,277.972,424.042,-179.928,13.923,150.874
C00687=1107.145,277.723,424.070,-179.932,13.921,150.874
C00688=1107.139,277.475,424.099,-179.936,13.921,150.875
C00689=1107.134,277.227,424.128,-179.940,13.921,150.876
C00690=1107.128,276.978,424.157,-179.944,13.921,150.877
C00691=1107.120,276.623,424.199,-179.950,13.920,150.878
C00692=1107.112,276.269,424.240,-179.955,13.920,150.879
C00693=1107.104,275.913,424.281,-179.961,13.919,150.880
C00694=1107.096,275.558,424.322,-179.966,13.919,150.882
C00695=1107.090,275.309,424.352,-179.970,13.919,150.883
C00696=1107.085,275.061,424.380,-179.974,13.919,150.883
C00697=1107.079,274.813,424.409,-179.977,13.919,150.884
C00698=1107.073,274.564,424.438,-179.982,13.918,150.885
C00699=1107.068,274.317,424.466,-179.986,13.918,150.886
C00700=1107.061,274.069,424.495,-179.990,13.918,150.887
C00701=1107.056,273.820,424.524,-179.993,13.917,150.887
C00702=1107.051,273.572,424.553,-179.997,13.917,150.888
C00703=1107.045,273.323,424.581,179.999,13.917,150.889
C00704=1107.038,273.075,424.610,179.995,13.917,150.890
C00705=1107.033,272.827,424.638,179.990,13.916,150.891
C00706=1107.028,272.578,424.667,179.987,13.916,150.892
C00707=1107.022,272.330,424.696,179.983,13.916,150.893
C00708=1107.016,272.082,424.724,179.979,13.915,150.893
C00709=1107.010,271.834,424.753,179.975,13.915,150.894
C00710=1107.005,271.585,424.782,179.971,13.915,150.895
C00711=1106.999,271.337,424.811,179.968,13.915,150.896
C00712=1106.993,271.089,424.839,179.964,13.915,150.897
C00713=1106.988,270.841,424.867,179.959,13.914,150.898
C00714=1106.982,270.592,424.896,179.955,13.914,150.898
C00715=1106.976,270.344,424.924,179.951,13.914,150.899
C00716=1106.971,270.095,424.953,179.947,13.914,150.900
C00717=1106.965,269.847,424.982,179.944,13.914,150.901
C00718=1106.959,269.599,425.010,179.940,13.914,150.902
C00719=1106.954,269.350,425.038,179.936,13.913,150.903
C00720=1106.948,269.102,425.066,179.932,13.913,150.903
C00721=1106.942,268.854,425.095,179.928,13.913,150.904
C00722=1106.937,268.606,425.123,179.925,13.913,150.905
C00723=1106.931,268.357,425.152,179.920,13.912,150.906
C00724=1106.925,268.109,425.180,179.916,13.912,150.907
C00725=1106.919,267.861,425.209,179.912,13.912,150.908
C00726=1106.913,267.612,425.237,179.908,13.912,150.909
C00727=1106.908,267.364,425.265,179.904,13.912,150.909
C00728=1106.902,267.116,425.293,179.901,13.912,150.910
C00729=1106.897,266.867,425.322,179.897,13.912,150.911
C00730=1106.891,266.618,425.350,179.893,13.912,150.912
C00731=1106.886,266.371,425.379,179.889,13.912,150.913
C00732=1106.880,266.122,425.407,179.885,13.912,150.914
C00733=1106.874,265.874,425.435,179.881,13.912,150.915
C00734=1106.868,265.626,425.463,179.877,13.912,150.916
C00735=1106.863,265.377,425.491,179.873,13.911,150.916
C00736=1106.857,265.129,425.520,179.869,13.911,150.917
C00737=1106.852,264.881,425.548,179.865,13.911,150.918
C00738=1106.846,264.632,425.576,179.861,13.911,150.919
C00739=1106.840,264.384,425.603,179.857,13.911,150.920
C00740=1106.834,264.135,425.632,179.853,13.911,150.921
C00741=1106.828,263.887,425.659,179.849,13.911,150.922
C00742=1106.823,263.639,425.688,179.845,13.911,150.923
C00743=1106.815,263.286,425.728,179.840,13.911,150.924
C00744=1106.807,262.934,425.767,179.834,13.910,150.925
C00745=1106.798,262.583,425.807,179.828,13.911,150.927
C00746=1106.790,262.229,425.846,179.823,13.911,150.928
C00747=1106.784,261.981,425.874,179.819,13.911,150.929
C00748=1106.779,261.733,425.902,179.815,13.911,150.930
C00749=1106.772,261.485,425.930,179.811,13.911,150.931
C00750=1106.767,261.237,425.958,179.807,13.911,150.931
C00751=1106.761,260.988,425.986,179.802,13.910,150.932
C00752=1106.756,260.740,426.014,179.799,13.910,150.933
C00753=1106.749,260.491,426.041,179.794,13.910,150.934
C00754=1106.744,260.243,426.069,179.791,13.910,150.935
C00755=1106.738,259.994,426.097,179.787,13.910,150.936
C00756=1106.733,259.746,426.125,179.783,13.910,150.937
C00757=1106.727,259.498,426.153,179.779,13.910,150.938
C00758=1106.721,259.249,426.180,179.775,13.910,150.939
C00759=1106.716,259.001,426.208,179.771,13.910,150.940
C00760=1106.710,258.752,426.237,179.767,13.910,150.940
C00761=1106.704,258.504,426.264,179.763,13.910,150.941
C00762=1106.699,258.255,426.291,179.759,13.910,150.942
C00763=1106.693,258.007,426.320,179.755,13.910,150.943
C00764=1106.687,257.759,426.347,179.751,13.910,150.944
C00765=1106.681,257.510,426.375,179.747,13.910,150.945
C00766=1106.676,257.262,426.403,179.743,13.910,150.946
C00767=1106.669,257.014,426.430,179.739,13.910,150.947
C00768=1106.664,256.764,426.457,179.735,13.911,150.948
C00769=1106.659,256.516,426.485,179.731,13.911,150.949
C00770=1106.653,256.268,426.512,179.727,13.910,150.950
C00771=1106.647,256.019,426.540,179.723,13.910,150.950
C00772=1106.641,255.772,426.568,179.720,13.910,150.951
C00773=1106.636,255.523,426.595,179.715,13.911,150.952
C00774=1106.630,255.274,426.623,179.711,13.911,150.953
C00775=1106.624,255.026,426.650,179.708,13.911,150.954
C00776=1106.619,254.778,426.678,179.704,13.911,150.955
C00777=1106.613,254.529,426.705,179.699,13.911,150.956
C00778=1106.607,254.281,426.733,179.696,13.911,150.957
C00779=1106.602,254.032,426.760,179.692,13.911,150.958
C00780=1106.596,253.784,426.788,179.688,13.911,150.959
C00781=1106.590,253.535,426.815,179.684,13.911,150.960
C00782=1106.584,253.287,426.842,179.680,13.911,150.961
C00783=1106.579,253.038,426.870,179.676,13.911,150.961
C00784=1106.573,252.790,426.896,179.672,13.911,150.962
C00785=1106.567,252.541,426.925,179.668,13.911,150.963
C00786=1106.562,252.293,426.951,179.664,13.911,150.964
C00787=1106.556,252.045,426.979,179.660,13.911,150.965
C00788=1106.550,251.797,427.006,179.656,13.911,150.966
C00789=1106.545,251.548,427.033,179.652,13.912,150.967
C00790=1106.539,251.299,427.061,179.648,13.912,150.968
C00791=1106.534,251.051,427.088,179.644,13.912,150.969
C00792=1106.528,250.802,427.115,179.640,13.912,150.970
C00793=1106.523,250.554,427.142,179.636,13.912,150.971
C00794=1106.516,250.305,427.170,179.632,13.912,150.972
C00795=1106.509,249.950,427.208,179.626,13.912,150.973
C00796=1106.501,249.595,427.248,179.620,13.912,150.974
C00797=1106.493,249.240,427.286,179.615,13.912,150.976
C00798=1106.485,248.885,427.324,179.609,13.912,150.977
C00799=1106.479,248.637,427.352,179.605,13.913,150.978
C00800=1106.473,248.388,427.379,179.601,13.913,150.979
C00801=1106.468,248.139,427.406,179.597,13.913,150.980
C00802=1106.462,247.891,427.433,179.594,13.913,150.981
C00803=1106.457,247.643,427.460,179.589,13.913,150.982
C00804=1106.452,247.394,427.487,179.585,13.913,150.983
C00805=1106.445,247.146,427.514,179.582,13.913,150.983
C00806=1106.439,246.897,427.541,179.577,13.913,150.984
C00807=1106.434,246.649,427.568,179.573,13.913,150.985
C00808=1106.428,246.400,427.595,179.569,13.914,150.986
C00809=1106.423,246.152,427.622,179.565,13.914,150.987
C00810=1106.417,245.903,427.649,179.561,13.914,150.988
C00811=1106.412,245.655,427.676,179.557,13.914,150.989
C00812=1106.406,245.407,427.702,179.553,13.914,150.990
C00813=1106.400,245.158,427.729,179.549,13.914,150.991
C00814=1106.395,244.909,427.757,179.546,13.915,150.992
C00815=1106.389,244.660,427.783,179.542,13.915,150.993
C00816=1106.383,244.412,427.810,179.538,13.915,150.994
C00817=1106.377,244.164,427.837,179.534,13.915,150.995
C00818=1106.372,243.915,427.864,179.530,13.915,150.996
C00819=1106.366,243.667,427.890,179.526,13.916,150.997
C00820=1106.361,243.418,427.917,179.522,13.916,150.998
C00821=1106.355,243.170,427.944,179.518,13.916,150.999
C00822=1106.349,242.922,427.970,179.514,13.916,151.000
C00823=1106.344,242.673,427.998,179.510,13.916,151.001
C00824=1106.339,242.424,428.024,179.506,13.916,151.002
C00825=1106.333,242.176,428.050,179.501,13.917,151.003
C00826=1106.326,241.927,428.077,179.498,13.917,151.003
C00827=1106.321,241.678,428.104,179.494,13.917,151.004
C00828=1106.315,241.430,428.130,179.489,13.917,151.005
C00829=1106.309,241.181,428.157,179.485,13.917,151.006
C00830=1106.304,240.932,428.183,179.482,13.918,151.007
C00831=1106.298,240.684,428.210,179.478,13.918,151.008
C00832=1106.292,240.436,428.236,179.474,13.919,151.009
C00833=1106.286,240.187,428.263,179.470,13.919,151.010
C00834=1106.281,239.939,428.290,179.466,13.919,151.011
C00835=1106.275,239.690,428.316,179.462,13.919,151.012
C00836=1106.269,239.442,428.342,179.458,13.919,151.013
C00837=1106.264,239.193,428.369,179.454,13.919,151.014
C00838=1106.258,238.944,428.395,179.449,13.920,151.015
C00839=1106.252,238.696,428.421,179.446,13.920,151.016
C00840=1106.247,238.448,428.448,179.441,13.920,151.017
C00841=1106.241,238.199,428.474,179.438,13.921,151.018
C00842=1106.235,237.950,428.501,179.434,13.921,151.019
C00843=1106.229,237.702,428.527,179.430,13.921,151.020
C00844=1106.224,237.453,428.553,179.426,13.922,151.021
C00845=1106.218,237.205,428.580,179.422,13.922,151.022
C00846=1106.212,236.956,428.607,179.418,13.922,151.023
C00847=1106.205,236.595,428.645,179.412,13.923,151.024
C00848=1106.196,236.233,428.683,179.406,13.923,151.026
C00849=1106.188,235.871,428.721,179.400,13.923,151.027
C00850=1106.180,235.509,428.760,179.394,13.923,151.029
C00851=1106.174,235.260,428.786,179.390,13.923,151.029
C00852=1106.169,235.012,428.812,179.386,13.924,151.030
C00853=1106.163,234.764,428.838,179.383,13.925,151.032
C00854=1106.157,234.515,428.864,179.379,13.925,151.032
C00855=1106.152,234.266,428.890,179.375,13.925,151.033
C00856=1106.146,234.018,428.916,179.371,13.925,151.034
C00857=1106.140,233.769,428.943,179.366,13.926,151.035
C00858=1106.135,233.520,428.969,179.363,13.926,151.036
C00859=1106.129,233.271,428.995,179.358,13.926,151.037
C00860=1106.123,233.023,429.021,179.354,13.926,151.038
C00861=1106.117,232.774,429.047,179.351,13.927,151.039
C00862=1106.112,232.527,429.073,179.347,13.927,151.040
C00863=1106.107,232.278,429.099,179.343,13.928,151.041
C00864=1106.101,232.029,429.124,179.339,13.928,151.042
C00865=1106.095,231.780,429.151,179.335,13.928,151.043
C00866=1106.089,231.532,429.177,179.330,13.929,151.044
C00867=1106.084,231.283,429.203,179.327,13.929,151.045
C00868=1106.078,231.034,429.230,179.322,13.929,151.046
C00869=1106.072,230.786,429.254,179.319,13.930,151.047
C00870=1106.067,230.537,429.280,179.315,13.930,151.048
C00871=1106.061,230.289,429.307,179.311,13.931,151.049
C00872=1106.055,230.040,429.332,179.307,13.931,151.050
C00873=1106.050,229.791,429.358,179.303,13.931,151.051
C00874=1106.044,229.542,429.384,179.299,13.931,151.052
C00875=1106.038,229.294,429.410,179.294,13.931,151.053
C00876=1106.033,229.046,429.436,179.291,13.933,151.054
C00877=1106.027,228.797,429.462,179.287,13.933,151.055
C00878=1106.021,228.548,429.487,179.283,13.933,151.056
C00879=1106.016,228.299,429.513,179.279,13.933,151.057
C00880=1106.009,228.051,429.538,179.275,13.933,151.058
C00881=1106.004,227.802,429.565,179.270,13.934,151.059
C00882=1105.999,227.554,429.591,179.267,13.935,151.060
C00883=1105.992,227.305,429.616,179.263,13.935,151.061
C00884=1105.987,227.056,429.642,179.259,13.935,151.062
C00885=1105.981,226.808,429.667,179.255,13.935,151.063
C00886=1105.975,226.559,429.693,179.251,13.936,151.064
C00887=1105.970,226.311,429.718,179.246,13.936,151.065
C00888=1105.964,226.062,429.744,179.243,13.937,151.066
C00889=1105.959,225.813,429.770,179.239,13.937,151.067
C00890=1105.953,225.564,429.795,179.235,13.938,151.068
C00891=1105.948,225.316,429.821,179.231,13.938,151.069
C00892=1105.942,225.067,429.846,179.227,13.938,151.070
C00893=1105.936,224.818,429.872,179.223,13.938,151.071
C00894=1105.930,224.569,429.898,179.219,13.939,151.072
C00895=1105.925,224.321,429.923,179.215,13.940,151.073
C00896=1105.919,224.073,429.948,179.211,13.940,151.074
C00897=1105.913,223.824,429.974,179.207,13.940,151.075
C00898=1105.908,223.576,429.999,179.203,13.941,151.076
C00899=1105.899,223.205,430.038,179.197,13.941,151.078
C00900=1105.890,222.835,430.075,179.191,13.942,151.079
C00901=1105.883,222.466,430.114,179.185,13.943,151.081
C00902=1105.874,222.095,430.151,179.180,13.944,151.082
C00903=1105.868,221.847,430.176,179.175,13.944,151.083
C00904=1105.862,221.598,430.202,179.171,13.945,151.084
C00905=1105.857,221.349,430.228,179.167,13.945,151.085
C00906=1105.851,221.101,430.252,179.163,13.945,151.086
C00907=1105.845,220.852,430.277,179.159,13.946,151.087
C00908=1105.840,220.603,430.303,179.156,13.946,151.088
C00909=1105.834,220.355,430.328,179.151,13.947,151.089
C00910=1105.828,220.106,430.353,179.147,13.947,151.090
C00911=1105.823,219.857,430.379,179.143,13.947,151.091
C00912=1105.817,219.609,430.404,179.140,13.948,151.092
C00913=1105.811,219.360,430.429,179.135,13.949,151.093
C00914=1105.805,219.111,430.455,179.131,13.949,151.094
C00915=1105.800,218.862,430.479,179.127,13.949,151.095
C00916=1105.794,218.614,430.505,179.123,13.950,151.096
C00917=1105.788,218.365,430.530,179.120,13.951,151.097
C00918=1105.783,218.116,430.555,179.116,13.951,151.098
C00919=1105.777,217.868,430.580,179.111,13.951,151.099
C00920=1105.771,217.620,430.605,179.107,13.952,151.100
C00921=1105.765,217.370,430.630,179.103,13.952,151.101
C00922=1105.760,217.121,430.656,179.100,13.953,151.102
C00923=1105.755,216.873,430.680,179.095,13.953,151.103
C00924=1105.748,216.624,430.705,179.091,13.954,151.104
C00925=1105.743,216.376,430.730,179.087,13.954,151.105
C00926=1105.738,216.127,430.755,179.084,13.955,151.106
C00927=1105.732,215.879,430.780,179.080,13.955,151.107
C00928=1105.726,215.629,430.805,179.076,13.956,151.108
C00929=1105.720,215.381,430.830,179.071,13.956,151.109
C00930=1105.715,215.132,430.855,179.067,13.956,151.111
C00931=1105.709,214.883,430.880,179.064,13.958,151.112
C00932=1105.704,214.634,430.905,179.060,13.958,151.112
C00933=1105.698,214.386,430.930,179.056,13.958,151.114
C00934=1105.692,214.137,430.954,179.051,13.959,151.115
C00935=1105.686,213.889,430.980,179.048,13.959,151.116
C00936=1105.681,213.640,431.004,179.044,13.960,151.117
C00937=1105.675,213.391,431.030,179.040,13.960,151.118
C00938=1105.670,213.142,431.054,179.036,13.960,151.119
C00939=1105.664,212.894,431.079,179.032,13.961,151.120
C00940=1105.659,212.645,431.104,179.028,13.962,151.121
C00941=1105.653,212.396,431.128,179.024,13.962,151.122
C00942=1105.647,212.148,431.153,179.020,13.962,151.123
C00943=1105.641,211.899,431.178,179.016,13.963,151.124
C00944=1105.636,211.651,431.203,179.012,13.964,151.125
C00945=1105.630,211.401,431.228,179.008,13.965,151.126
C00946=1105.624,211.153,431.252,179.004,13.965,151.127
C00947=1105.618,210.904,431.277,179.000,13.965,151.128
C00948=1105.613,210.655,431.301,178.996,13.966,151.129
C00949=1105.607,210.406,431.326,178.992,13.967,151.130
C00950=1105.602,210.158,431.350,178.988,13.967,151.131
C00951=1105.593,209.791,431.387,178.982,13.968,151.132
C00952=1105.584,209.424,431.423,178.976,13.968,151.134
C00953=1105.577,209.058,431.460,178.970,13.970,151.135
C00954=1105.568,208.691,431.496,178.965,13.970,151.137
C00955=1105.545,207.696,431.593,178.940,13.971,151.143
C00956=1105.539,207.447,431.618,178.936,13.973,151.144
C00957=1105.534,207.198,431.642,178.931,13.974,151.145
C00958=1105.528,206.949,431.667,178.927,13.976,151.147
C00959=1105.522,206.701,431.691,178.922,13.977,151.148
C00960=1105.516,206.451,431.715,178.918,13.978,151.149
C00961=1105.511,206.203,431.740,178.914,13.979,151.150
C00962=1105.505,205.954,431.764,178.910,13.981,151.152
C00963=1105.499,205.705,431.788,178.906,13.982,151.153
C00964=1105.493,205.457,431.812,178.901,13.984,151.154
C00965=1105.488,205.208,431.836,178.897,13.985,151.156
C00966=1105.482,204.959,431.861,178.893,13.986,151.157
C00967=1105.477,204.710,431.885,178.889,13.988,151.158
C00968=1105.471,204.462,431.909,178.884,13.989,151.159
C00969=1105.465,204.213,431.934,178.881,13.990,151.161
C00970=1105.460,203.964,431.958,178.876,13.991,151.162
C00971=1105.454,203.716,431.982,178.872,13.993,151.163
C00972=1105.448,203.467,432.006,178.868,13.994,151.164
C00973=1105.442,203.218,432.030,178.864,13.995,151.166
C00974=1105.437,202.969,432.055,178.859,13.996,151.167
C00975=1105.431,202.720,432.079,178.855,13.998,151.168
C00976=1105.425,202.472,432.103,178.850,13.999,151.169
C00977=1105.419,202.223,432.127,178.846,14.001,151.171
C00978=1105.413,201.974,432.151,178.842,14.002,151.172
C00979=1105.408,201.726,432.175,178.838,14.003,151.173
C00980=1105.402,201.476,432.199,178.833,14.004,151.174
C00981=1105.396,201.227,432.223,178.830,14.006,151.176
C00982=1105.390,200.979,432.247,178.826,14.007,151.177
C00983=1105.384,200.730,432.271,178.821,14.008,151.178
C00984=1105.378,200.482,432.295,178.817,14.010,151.179
C00985=1105.373,200.233,432.319,178.813,14.011,151.181
C00986=1105.367,199.983,432.342,178.808,14.013,151.182
C00987=1105.361,199.735,432.367,178.804,14.014,151.183
C00988=1105.355,199.487,432.390,178.800,14.015,151.185
C00989=1105.350,199.238,432.415,178.795,14.016,151.186
C00990=1105.345,198.988,432.439,178.792,14.018,151.187
C00991=1105.339,198.740,432.462,178.787,14.019,151.188
C00992=1105.332,198.492,432.486,178.783,14.021,151.189
C00993=1105.327,198.243,432.510,178.779,14.021,151.191
C00994=1105.321,197.993,432.533,178.775,14.023,151.192
C00995=1105.316,197.745,432.558,178.770,14.024,151.193
C00996=1105.310,197.496,432.581,178.766,14.026,151.194
C00997=1105.305,197.247,432.605,178.762,14.027,151.196
C00998=1105.298,196.998,432.629,178.758,14.028,151.197
C00999=1105.293,196.750,432.653,178.754,14.029,151.198
C01000=1105.287,196.501,432.676,178.750,14.030,151.199
C01001=1105.282,196.252,432.700,178.746,14.032,151.201
C01002=1105.275,196.003,432.724,178.741,14.033,151.202
C01003=1105.270,195.754,432.748,178.737,14.035,151.203
C01004=1105.264,195.506,432.772,178.733,14.035,151.204
C01005=1105.258,195.257,432.795,178.729,14.037,151.205
C01006=1105.253,195.008,432.819,178.724,14.038,151.207
C01007=1105.247,194.759,432.842,178.721,14.040,151.208
C01008=1105.241,194.510,432.866,178.716,14.040,151.209
C01009=1105.236,194.261,432.889,178.713,14.042,151.210
C01010=1105.229,194.013,432.913,178.708,14.043,151.212
C01011=1105.224,193.764,432.937,178.704,14.044,151.213
C01012=1105.218,193.515,432.960,178.699,14.045,151.214
C01013=1105.213,193.266,432.984,178.696,14.047,151.215
C01014=1105.207,193.017,433.008,178.692,14.048,151.216
C01015=1105.201,192.768,433.031,178.688,14.049,151.218
C01016=1105.195,192.497,433.056,178.683,14.051,151.219
C01017=1105.189,192.226,433.082,178.679,14.052,151.220
C01018=1105.183,191.956,433.108,178.674,14.053,151.222
C01019=1105.176,191.684,433.133,178.669,14.055,151.223
C01020=1105.171,191.436,433.156,178.665,14.056,151.224
C01021=1105.165,191.187,433.181,178.661,14.057,151.225
C01022=1105.160,190.938,433.204,178.657,14.058,151.226
C01023=1105.154,190.689,433.227,178.653,14.059,151.228
C01024=1105.148,190.441,433.251,178.649,14.061,151.229
C01025=1105.143,190.192,433.274,178.645,14.062,151.230
C01026=1105.137,189.943,433.297,178.641,14.063,151.231
C01027=1105.131,189.695,433.320,178.637,14.065,151.233
C01028=1105.126,189.445,433.344,178.633,14.065,151.234
C01029=1105.120,189.196,433.367,178.629,14.067,151.235
C01030=1105.115,188.948,433.390,178.624,14.068,151.236
C01031=1105.109,188.699,433.414,178.621,14.069,151.237
C01032=1105.103,188.449,433.437,178.616,14.070,151.238
C01033=1105.097,188.200,433.460,178.612,14.072,151.240
C01034=1105.091,187.952,433.483,178.608,14.072,151.241
C01035=1105.086,187.702,433.507,178.604,14.074,151.242
C01036=1105.080,187.454,433.530,178.600,14.075,151.243
C01037=1105.075,187.205,433.553,178.596,14.076,151.244
C01038=1105.069,186.956,433.576,178.592,14.077,151.246
C01039=1105.063,186.707,433.599,178.588,14.078,151.247
C01040=1105.058,186.458,433.623,178.583,14.079,151.248
C01041=1105.052,186.209,433.646,178.580,14.081,151.249
C01042=1105.047,185.962,433.669,178.575,14.082,151.250
C01043=1105.041,185.713,433.692,178.572,14.083,151.251
C01044=1105.036,185.464,433.715,178.567,14.084,151.253
C01045=1105.031,185.215,433.738,178.564,14.085,151.254
C01046=1105.025,184.966,433.761,178.560,14.087,151.255
C01047=1105.019,184.717,433.784,178.555,14.088,151.256
C01048=1105.013,184.467,433.808,178.552,14.089,151.257
C01049=1105.007,184.218,433.831,178.547,14.090,151.258
C01050=1105.001,183.970,433.853,178.543,14.092,151.260
C01051=1104.995,183.721,433.876,178.539,14.092,151.261
C01052=1104.989,183.472,433.899,178.535,14.094,151.262
C01053=1104.983,183.223,433.922,178.531,14.095,151.263
C01054=1104.978,182.974,433.945,178.527,14.096,151.264
C01055=1104.972,182.725,433.968,178.523,14.097,151.266
C01056=1104.966,182.476,433.991,178.519,14.098,151.267
C01057=1104.960,182.228,434.014,178.515,14.100,151.268
C01058=1104.955,181.979,434.037,178.511,14.101,151.269
C01059=1104.949,181.730,434.060,178.507,14.102,151.270
C01060=1104.943,181.481,434.082,178.503,14.103,151.271
C01061=1104.938,181.232,434.105,178.499,14.104,151.273
C01062=1104.931,180.983,434.128,178.494,14.105,151.274
C01063=1104.925,180.734,434.151,178.491,14.107,151.275
C01064=1104.920,180.486,434.174,178.486,14.108,151.276
C01065=1104.914,180.237,434.197,178.483,14.109,151.277
C01066=1104.909,179.988,434.219,178.478,14.110,151.278
C01067=1104.903,179.739,434.241,178.475,14.111,151.279
C01068=1104.898,179.490,434.264,178.471,14.113,151.281
C01069=1104.891,179.241,434.287,178.467,14.113,151.282
C01070=1104.885,178.993,434.310,178.463,14.115,151.283
C01071=1104.880,178.744,434.333,178.459,14.116,151.284
C01072=1104.874,178.495,434.356,178.455,14.117,151.285
C01073=1104.869,178.245,434.378,178.450,14.118,151.286
C01074=1104.863,177.996,434.401,178.447,14.119,151.288
C01075=1104.856,177.748,434.423,178.442,14.120,151.289
C01076=1104.851,177.499,434.446,178.439,14.121,151.290
C01077=1104.846,177.250,434.468,178.434,14.122,151.291
C01078=1104.840,177.001,434.491,178.431,14.124,151.292
C01079=1104.834,176.752,434.514,178.426,14.124,151.293
C01080=1104.828,176.481,434.538,178.423,14.126,151.295
C01081=1104.822,176.209,434.562,178.418,14.127,151.296
C01082=1104.816,175.938,434.587,178.413,14.128,151.297
C01083=1104.809,175.667,434.612,178.410,14.130,151.298
C01084=1104.803,175.417,434.634,178.405,14.130,151.299
C01085=1104.798,175.169,434.657,178.402,14.132,151.301
C01086=1104.792,174.920,434.680,178.397,14.132,151.302
C01087=1104.786,174.671,434.701,178.394,14.134,151.303
C01088=1104.780,174.422,434.724,178.389,14.135,151.304
C01089=1104.775,174.173,434.746,178.386,14.136,151.305
C01090=1104.770,173.924,434.769,178.382,14.137,151.306
C01091=1104.763,173.676,434.791,178.378,14.138,151.307
C01092=1104.758,173.426,434.814,178.374,14.139,151.308
C01093=1104.752,173.177,434.837,178.370,14.140,151.310
C01094=1104.746,172.928,434.858,178.366,14.141,151.311
C01095=1104.741,172.680,434.881,178.362,14.142,151.312
C01096=1104.735,172.430,434.903,178.358,14.144,151.313
C01097=1104.729,172.182,434.925,178.354,14.144,151.314
C01098=1104.724,171.932,434.948,178.350,14.145,151.315
C01099=1104.718,171.684,434.970,178.346,14.146,151.316
C01100=1104.712,171.435,434.992,178.343,14.147,151.317
C01101=1104.707,171.186,435.015,178.338,14.148,151.319
C01102=1104.701,170.937,435.037,178.335,14.150,151.320
C01103=1104.695,170.689,435.059,178.331,14.151,151.321
C01104=1104.690,170.439,435.081,178.327,14.151,151.322
C01105=1104.684,170.190,435.103,178.323,14.153,151.323
C01106=1104.678,169.941,435.126,178.319,14.153,151.324
C01107=1104.673,169.692,435.148,178.316,14.155,151.325
C01108=1104.667,169.444,435.170,178.311,14.155,151.326
C01109=1104.661,169.194,435.192,178.307,14.157,151.327
C01110=1104.656,168.945,435.214,178.303,14.158,151.328
C01111=1104.650,168.697,435.236,178.300,14.159,151.329
C01112=1104.644,168.447,435.259,178.295,14.159,151.331
C01113=1104.639,168.199,435.280,178.292,14.161,151.332
C01114=1104.633,167.950,435.303,178.288,14.161,151.333
C01115=1104.628,167.700,435.325,178.284,14.163,151.334
C01116=1104.622,167.452,435.346,178.281,14.164,151.335
C01117=1104.617,167.202,435.369,178.276,14.164,151.336
C01118=1104.610,166.954,435.391,178.273,14.166,151.337
C01119=1104.605,166.705,435.413,178.269,14.166,151.338
C01120=1104.599,166.456,435.434,178.265,14.168,151.339
C01121=1104.594,166.206,435.457,178.261,14.168,151.340
C01122=1104.588,165.958,435.479,178.257,14.170,151.341
C01123=1104.583,165.709,435.501,178.253,14.170,151.342
C01124=1104.577,165.460,435.522,178.250,14.171,151.344
C01125=1104.572,165.211,435.544,178.245,14.172,151.345
C01126=1104.565,164.962,435.566,178.242,14.173,151.346
C01127=1104.560,164.713,435.589,178.238,14.174,151.347
C01128=1104.554,164.464,435.610,178.234,14.175,151.348
C01129=1104.549,164.215,435.632,178.231,14.176,151.349
C01130=1104.543,163.966,435.654,178.227,14.177,151.350
C01131=1104.538,163.717,435.676,178.223,14.178,151.351
C01132=1104.532,163.468,435.697,178.219,14.179,151.352
C01133=1104.527,163.219,435.719,178.215,14.180,151.353
C01134=1104.521,162.970,435.741,178.211,14.180,151.354
C01135=1104.515,162.721,435.764,178.208,14.181,151.355
C01136=1104.510,162.473,435.785,178.204,14.182,151.356
C01137=1104.504,162.223,435.807,178.200,14.183,151.357
C01138=1104.499,161.975,435.828,178.196,14.184,151.358
C01139=1104.493,161.725,435.851,178.193,14.185,151.359
C01140=1104.488,161.477,435.872,178.188,14.186,151.360
C01141=1104.482,161.227,435.894,178.185,14.187,151.361
C01142=1104.476,160.978,435.916,178.182,14.188,151.362
C01143=1104.471,160.729,435.937,178.177,14.189,151.364
C01144=1104.464,160.457,435.960,178.173,14.190,151.365
C01145=1104.458,160.185,435.984,178.169,14.191,151.366
C01146=1104.452,159.914,436.008,178.165,14.192,151.367
C01147=1104.446,159.642,436.031,178.160,14.193,151.368
C01148=1104.440,159.393,436.053,178.157,14.194,151.369
C01149=1104.434,159.144,436.075,178.154,14.195,151.370
C01150=1104.428,158.896,436.096,178.149,14.195,151.371
C01151=1104.423,158.646,436.118,178.146,14.197,151.372
C01152=1104.418,158.397,436.139,178.142,14.197,151.373
C01153=1104.411,158.148,436.160,178.138,14.199,151.375
C01154=1104.406,157.899,436.182,178.134,14.199,151.375
C01155=1104.400,157.650,436.204,178.131,14.200,151.377
C01156=1104.395,157.401,436.225,178.127,14.201,151.378
C01157=1104.389,157.152,436.247,178.123,14.202,151.379
C01158=1104.383,156.903,436.268,178.119,14.202,151.380
C01159=1104.377,156.654,436.289,178.116,14.204,151.381
C01160=1104.372,156.405,436.310,178.112,14.205,151.382
C01161=1104.366,156.156,436.332,178.108,14.205,151.383
C01162=1104.361,155.907,436.354,178.105,14.206,151.384
C01163=1104.355,155.658,436.375,178.100,14.207,151.385
C01164=1104.349,155.409,436.396,178.097,14.208,151.386
C01165=1104.343,155.160,436.417,178.093,14.209,151.387
C01166=1104.338,154.911,436.439,178.089,14.210,151.388
C01167=1104.331,154.662,436.460,178.086,14.210,151.389
C01168=1104.326,154.413,436.481,178.082,14.211,151.390
C01169=1104.321,154.164,436.502,178.079,14.213,151.391
C01170=1104.315,153.915,436.524,178.075,14.213,151.392
C01171=1104.310,153.666,436.545,178.071,14.214,151.393
C01172=1104.304,153.416,436.567,178.067,14.215,151.394
C01173=1104.298,153.168,436.588,178.064,14.216,151.395
C01174=1104.292,152.918,436.609,178.059,14.216,151.396
C01175=1104.287,152.670,436.630,178.056,14.217,151.397
C01176=1104.281,152.421,436.651,178.052,14.218,151.398
C01177=1104.275,152.171,436.672,178.049,14.219,151.399
C01178=1104.270,151.923,436.694,178.045,14.220,151.400
C01179=1104.264,151.674,436.715,178.041,14.221,151.401
C01180=1104.258,151.424,436.736,178.038,14.222,151.402
C01181=1104.252,151.175,436.757,178.034,14.222,151.403
C01182=1104.247,150.926,436.778,178.031,14.223,151.404
C01183=1104.241,150.678,436.799,178.026,14.224,151.405
C01184=1104.235,150.428,436.820,178.023,14.225,151.406
C01185=1104.230,150.179,436.841,178.019,14.225,151.407
C01186=1104.225,149.930,436.862,178.016,14.226,151.408
C01187=1104.219,149.681,436.884,178.011,14.227,151.409
C01188=1104.213,149.432,436.904,178.008,14.228,151.410
C01189=1104.207,149.183,436.926,178.005,14.229,151.411
C01190=1104.202,148.933,436.946,178.001,14.229,151.412
C01191=1104.196,148.685,436.968,177.997,14.231,151.413
C01192=1104.190,148.435,436.988,177.993,14.231,151.414
C01193=1104.184,148.187,437.009,177.990,14.232,151.415
C01194=1104.179,147.938,437.030,177.986,14.232,151.416
C01195=1104.173,147.689,437.051,177.982,14.234,151.417
C01196=1104.167,147.439,437.072,177.979,14.235,151.418
C01197=1104.162,147.191,437.093,177.975,14.235,151.419
C01198=1104.156,146.941,437.114,177.972,14.236,151.420
C01199=1104.150,146.692,437.134,177.968,14.236,151.421
C01200=1104.144,146.444,437.155,177.964,14.238,151.422
C01201=1104.139,146.194,437.176,177.961,14.238,151.423
C01202=1104.133,145.946,437.198,177.957,14.239,151.424
C01203=1104.128,145.696,437.218,177.953,14.239,151.425
C01204=1104.121,145.447,437.238,177.950,14.240,151.426
C01205=1104.116,145.198,437.260,177.946,14.242,151.427
C01206=1104.110,144.949,437.280,177.942,14.242,151.428
C01207=1104.105,144.699,437.301,177.939,14.243,151.429
C01208=1104.099,144.428,437.324,177.935,14.243,151.430
C01209=1104.092,144.156,437.346,177.931,14.244,151.431
C01210=1104.086,143.883,437.369,177.927,14.245,151.432
C01211=1104.080,143.612,437.392,177.923,14.246,151.433
C01212=1104.075,143.363,437.412,177.920,14.247,151.434
C01213=1104.068,143.113,437.433,177.916,14.247,151.435
C01214=1104.063,142.864,437.453,177.913,14.248,151.436
C01215=1104.057,142.616,437.474,177.909,14.249,151.437
C01216=1104.052,142.367,437.495,177.905,14.250,151.438
C01217=1104.045,142.117,437.515,177.901,14.250,151.439
C01218=1104.040,141.868,437.536,177.898,14.251,151.440
C01219=1104.035,141.619,437.556,177.894,14.252,151.441
C01220=1104.029,141.370,437.578,177.891,14.252,151.442
C01221=1104.023,141.121,437.598,177.888,14.253,151.443
C01222=1104.017,140.872,437.619,177.884,14.254,151.444
C01223=1104.012,140.623,437.639,177.881,14.254,151.444
C01224=1104.006,140.374,437.659,177.876,14.255,151.446
C01225=1104.001,140.125,437.680,177.873,14.256,151.446
C01226=1103.995,139.875,437.701,177.869,14.256,151.447
C01227=1103.989,139.626,437.720,177.866,14.257,151.448
C01228=1103.983,139.377,437.742,177.863,14.258,151.449
C01229=1103.977,139.129,437.762,177.859,14.258,151.450
C01230=1103.972,138.879,437.782,177.855,14.260,151.451
C01231=1103.966,138.630,437.803,177.852,14.260,151.452
C01232=1103.960,138.381,437.823,177.848,14.261,151.453
C01233=1103.955,138.132,437.844,177.844,14.261,151.454
C01234=1103.949,137.883,437.864,177.841,14.262,151.455
C01235=1103.944,137.634,437.884,177.837,14.262,151.456
C01236=1103.937,137.384,437.905,177.834,14.263,151.457
C01237=1103.932,137.135,437.925,177.831,14.264,151.458
C01238=1103.926,136.886,437.945,177.827,14.265,151.459
C01239=1103.921,136.637,437.966,177.824,14.266,151.460
C01240=1103.915,136.388,437.986,177.820,14.266,151.461
C01241=1103.910,136.139,438.006,177.816,14.267,151.461
C01242=1103.904,135.890,438.026,177.813,14.267,151.462
C01243=1103.898,135.641,438.047,177.809,14.268,151.463
C01244=1103.892,135.391,438.066,177.806,14.269,151.464
C01245=1103.887,135.142,438.087,177.802,14.269,151.465
C01246=1103.881,134.893,438.107,177.799,14.270,151.466
C01247=1103.875,134.644,438.127,177.795,14.270,151.467
C01248=1103.870,134.395,438.147,177.792,14.271,151.468
C01249=1103.864,134.146,438.168,177.788,14.271,151.469
C01250=1103.858,133.897,438.188,177.785,14.272,151.470
C01251=1103.852,133.648,438.209,177.782,14.273,151.471
C01252=1103.847,133.398,438.228,177.778,14.274,151.472
C01253=1103.841,133.149,438.248,177.775,14.274,151.472
C01254=1103.835,132.900,438.268,177.771,14.275,151.473
C01255=1103.830,132.651,438.289,177.768,14.276,151.474
C01256=1103.824,132.402,438.309,177.764,14.275,151.475
C01257=1103.819,132.153,438.328,177.761,14.276,151.476
C01258=1103.813,131.904,438.349,177.758,14.277,151.477
C01259=1103.807,131.655,438.369,177.754,14.277,151.478
C01260=1103.801,131.406,438.389,177.751,14.278,151.479
C01261=1103.796,131.156,438.409,177.747,14.279,151.480
C01262=1103.790,130.907,438.429,177.743,14.280,151.481
C01263=1103.784,130.658,438.449,177.740,14.280,151.482
C01264=1103.778,130.409,438.469,177.736,14.281,151.482
C01265=1103.773,130.159,438.489,177.733,14.282,151.483
C01266=1103.767,129.911,438.509,177.729,14.282,151.484
C01267=1103.761,129.662,438.529,177.726,14.283,151.485
C01268=1103.756,129.412,438.548,177.722,14.283,151.486
C01269=1103.750,129.163,438.568,177.719,14.284,151.487
C01270=1103.744,128.914,438.588,177.715,14.284,151.488
C01271=1103.738,128.665,438.608,177.712,14.285,151.489
C01272=1103.731,128.393,438.630,177.708,14.285,151.490
C01273=1103.726,128.121,438.652,177.705,14.286,151.491
C01274=1103.720,127.849,438.673,177.701,14.287,151.492
C01275=1103.713,127.576,438.695,177.697,14.287,151.493
C01276=1103.707,127.327,438.715,177.694,14.288,151.493
C01277=1103.701,127.078,438.734,177.691,14.289,151.494
C01278=1103.696,126.829,438.754,177.687,14.289,151.495
C01279=1103.690,126.579,438.774,177.684,14.290,151.496
C01280=1103.684,126.331,438.794,177.680,14.290,151.497
C01281=1103.679,126.081,438.813,177.677,14.291,151.498
C01282=1103.673,125.832,438.833,177.673,14.291,151.499
C01283=1103.668,125.583,438.853,177.670,14.292,151.500
C01284=1103.662,125.334,438.873,177.667,14.292,151.500
C01285=1103.656,125.084,438.892,177.663,14.293,151.501
C01286=1103.650,124.836,438.912,177.660,14.293,151.502
C01287=1103.644,124.586,438.931,177.656,14.293,151.503
C01288=1103.638,124.337,438.951,177.653,14.294,151.504
C01289=1103.633,124.088,438.971,177.650,14.295,151.505
C01290=1103.627,123.839,438.991,177.646,14.295,151.506
C01291=1103.622,123.590,439.010,177.643,14.296,151.507
C01292=1103.617,123.341,439.029,177.639,14.296,151.507
C01293=1103.611,123.092,439.049,177.636,14.297,151.508
C01294=1103.605,122.842,439.068,177.632,14.297,151.509
C01295=1103.599,122.594,439.088,177.629,14.298,151.510
C01296=1103.593,122.344,439.107,177.626,14.299,151.511
C01297=1103.588,122.094,439.127,177.623,14.298,151.512
C01298=1103.582,121.846,439.147,177.620,14.299,151.512
C01299=1103.577,121.596,439.166,177.616,14.300,151.513
C01300=1103.571,121.347,439.186,177.613,14.300,151.514
C01301=1103.565,121.098,439.206,177.609,14.300,151.515
C01302=1103.560,120.849,439.225,177.606,14.301,151.516
C01303=1103.554,120.600,439.244,177.603,14.302,151.517
C01304=1103.548,120.351,439.264,177.599,14.302,151.518
C01305=1103.543,120.102,439.283,177.596,14.303,151.518
C01306=1103.537,119.852,439.302,177.592,14.302,151.519
C01307=1103.531,119.603,439.321,177.589,14.303,151.520
C01308=1103.525,119.354,439.341,177.586,14.304,151.521
C01309=1103.520,119.105,439.360,177.583,14.304,151.522
C01310=1103.514,118.856,439.380,177.580,14.305,151.523
C01311=1103.509,118.606,439.399,177.576,14.305,151.523
C01312=1103.503,118.357,439.419,177.573,14.305,151.524
C01313=1103.497,118.108,439.438,177.569,14.306,151.525
C01314=1103.491,117.859,439.457,177.566,14.306,151.526
C01315=1103.486,117.610,439.476,177.563,14.307,151.527
C01316=1103.481,117.360,439.495,177.559,14.307,151.528
C01317=1103.475,117.111,439.515,177.557,14.307,151.528
C01318=1103.469,116.862,439.535,177.553,14.308,151.529
C01319=1103.463,116.613,439.554,177.550,14.308,151.530
C01320=1103.458,116.364,439.573,177.546,14.308,151.531
C01321=1103.452,116.115,439.592,177.543,14.309,151.532
C01322=1103.447,115.865,439.611,177.540,14.310,151.532
C01323=1103.441,115.616,439.630,177.537,14.309,151.533
C01324=1103.436,115.367,439.649,177.533,14.310,151.534
C01325=1103.430,115.118,439.669,177.530,14.310,151.535
C01326=1103.425,114.868,439.688,177.527,14.311,151.536
C01327=1103.419,114.619,439.707,177.524,14.312,151.536
C01328=1103.413,114.371,439.727,177.520,14.312,151.537
C01329=1103.408,114.121,439.746,177.517,14.312,151.538
C01330=1103.402,113.872,439.765,177.513,14.312,151.539
C01331=1103.396,113.622,439.784,177.511,14.313,151.540
C01332=1103.391,113.374,439.803,177.507,14.313,151.540
C01333=1103.385,113.124,439.822,177.504,14.314,151.541
C01334=1103.379,112.875,439.841,177.501,14.314,151.542
C01335=1103.374,112.626,439.860,177.497,14.314,151.543
C01336=1103.368,112.353,439.881,177.494,14.315,151.544
C01337=1103.361,112.081,439.902,177.491,14.315,151.545
C01338=1103.355,111.809,439.922,177.487,14.315,151.545
C01339=1103.349,111.536,439.943,177.484,14.316,151.546
C01340=1103.344,111.287,439.962,177.480,14.316,151.547
C01341=1103.337,111.038,439.981,177.477,14.316,151.548
C01342=1103.332,110.789,440.000,177.473,14.317,151.549
C01343=1103.326,110.540,440.019,177.470,14.317,151.550
C01344=1103.320,110.291,440.037,177.467,14.318,151.550
C01345=1103.314,110.041,440.057,177.464,14.318,151.551
C01346=1103.309,109.792,440.076,177.461,14.319,151.552
C01347=1103.303,109.543,440.094,177.457,14.318,151.553
C01348=1103.297,109.293,440.113,177.454,14.319,151.554
C01349=1103.292,109.044,440.132,177.451,14.319,151.554
C01350=1103.286,108.795,440.150,177.448,14.319,151.555
C01351=1103.280,108.546,440.170,177.445,14.320,151.556
C01352=1103.274,108.296,440.189,177.441,14.320,151.557
C01353=1103.269,108.048,440.207,177.438,14.321,151.557
C01354=1103.263,107.798,440.226,177.435,14.321,151.558
C01355=1103.258,107.549,440.245,177.432,14.321,151.559
C01356=1103.252,107.300,440.263,177.429,14.321,151.560
C01357=1103.246,107.051,440.282,177.425,14.321,151.560
C01358=1103.241,106.801,440.301,177.423,14.322,151.561
C01359=1103.235,106.552,440.319,177.419,14.323,151.562
C01360=1103.229,106.303,440.338,177.416,14.323,151.563
C01361=1103.223,106.054,440.357,177.413,14.323,151.564
C01362=1103.218,105.804,440.375,177.409,14.323,151.564
C01363=1103.212,105.555,440.394,177.406,14.324,151.565
C01364=1103.206,105.306,440.413,177.404,14.324,151.566
C01365=1103.201,105.056,440.431,177.400,14.324,151.567
C01366=1103.195,104.807,440.450,177.397,14.324,151.567
C01367=1103.190,104.559,440.469,177.394,14.324,151.568
C01368=1103.184,104.309,440.487,177.391,14.325,151.569
C01369=1103.178,104.059,440.506,177.388,14.325,151.570
C01370=1103.173,103.811,440.525,177.384,14.325,151.570
C01371=1103.167,103.561,440.543,177.381,14.326,151.571
C01372=1103.161,103.312,440.562,177.378,14.326,151.572
C01373=1103.155,103.063,440.580,177.375,14.326,151.573
C01374=1103.150,102.814,440.598,177.372,14.327,151.573
C01375=1103.145,102.564,440.618,177.369,14.326,151.574
C01376=1103.138,102.315,440.636,177.366,14.327,151.575
C01377=1103.133,102.066,440.655,177.362,14.327,151.576
C01378=1103.127,101.816,440.672,177.359,14.327,151.576
C01379=1103.122,101.567,440.691,177.356,14.328,151.577
C01380=1103.116,101.318,440.709,177.353,14.327,151.578
C01381=1103.111,101.069,440.728,177.350,14.328,151.579
C01382=1103.105,100.820,440.747,177.347,14.328,151.579
C01383=1103.098,100.570,440.765,177.344,14.328,151.580
C01384=1103.093,100.321,440.784,177.341,14.329,151.581
C01385=1103.087,100.072,440.802,177.337,14.329,151.582
C01386=1103.082,99.823,440.820,177.335,14.329,151.582
C01387=1103.076,99.573,440.838,177.332,14.330,151.583
C01388=1103.070,99.325,440.857,177.328,14.330,151.584
C01389=1103.065,99.075,440.875,177.325,14.330,151.585
C01390=1103.059,98.825,440.893,177.322,14.330,151.585
C01391=1103.053,98.576,440.911,177.319,14.330,151.586
C01392=1103.047,98.326,440.930,177.316,14.331,151.587
C01393=1103.042,98.078,440.948,177.313,14.330,151.587
C01394=1103.036,97.828,440.967,177.310,14.331,151.588
C01395=1103.031,97.579,440.984,177.306,14.331,151.589
C01396=1103.024,97.330,441.003,177.304,14.331,151.590
C01397=1103.020,97.080,441.021,177.301,14.332,151.590
C01398=1103.013,96.831,441.040,177.297,14.331,151.591
C01399=1103.008,96.582,441.057,177.295,14.332,151.592
C01400=1103.001,96.310,441.077,177.291,14.332,151.593
C01401=1102.995,96.037,441.098,177.288,14.332,151.593
C01402=1102.989,95.765,441.117,177.284,14.333,151.594
C01403=1102.983,95.493,441.137,177.281,14.332,151.595
C01404=1102.977,95.243,441.155,177.278,14.332,151.596
C01405=1102.971,94.995,441.173,177.275,14.333,151.596
C01406=1102.966,94.745,441.191,177.272,14.333,151.597
C01407=1102.960,94.496,441.209,177.269,14.333,151.598
C01408=1102.954,94.247,441.228,177.266,14.333,151.598
C01409=1102.949,93.997,441.246,177.263,14.333,151.599
C01410=1102.943,93.748,441.263,177.260,14.334,151.600
C01411=1102.937,93.499,441.281,177.257,14.333,151.601
C01412=1102.932,93.250,441.300,177.254,14.334,151.601
C01413=1102.926,93.000,441.318,177.251,14.334,151.602
C01414=1102.921,92.751,441.336,177.248,14.334,151.603
C01415=1102.914,92.501,441.354,177.245,14.334,151.603
C01416=1102.909,92.252,441.371,177.241,14.334,151.604
C01417=1102.904,92.004,441.390,177.239,14.334,151.605
C01418=1102.898,91.754,441.408,177.236,14.335,151.606
C01419=1102.892,91.505,441.426,177.233,14.334,151.606
C01420=1102.886,91.255,441.444,177.230,14.335,151.607
C01421=1102.881,91.006,441.462,177.227,14.335,151.608
C01422=1102.876,90.757,441.479,177.224,14.335,151.608
C01423=1102.870,90.507,441.497,177.221,14.335,151.609
C01424=1102.864,90.259,441.515,177.217,14.335,151.610
C01425=1102.858,90.009,441.533,177.215,14.335,151.610
C01426=1102.852,89.760,441.551,177.212,14.336,151.611
C01427=1102.847,89.511,441.569,177.209,14.335,151.612
C01428=1102.841,89.261,441.586,177.206,14.336,151.612
C01429=1102.835,89.012,441.604,177.203,14.336,151.613
C01430=1102.829,88.762,441.622,177.200,14.336,151.614
C01431=1102.823,88.513,441.640,177.197,14.336,151.615
C01432=1102.817,88.263,441.657,177.193,14.336,151.615
C01433=1102.812,88.014,441.675,177.191,14.336,151.616
C01434=1102.806,87.765,441.693,177.188,14.336,151.616
C01435=1102.800,87.516,441.711,177.184,14.336,151.617
C01436=1102.795,87.267,441.728,177.182,14.337,151.618
C01437=1102.790,87.017,441.746,177.179,14.337,151.619
C01438=1102.784,86.767,441.764,177.176,14.337,151.619
C01439=1102.778,86.518,441.782,177.173,14.337,151.620
C01440=1102.773,86.269,441.799,177.170,14.337,151.621
C01441=1102.767,86.020,441.817,177.167,14.337,151.621
C01442=1102.761,85.771,441.835,177.164,14.337,151.622
C01443=1102.756,85.522,441.852,177.161,14.337,151.623
C01444=1102.749,85.272,441.870,177.158,14.337,151.623
C01445=1102.744,85.023,441.888,177.155,14.337,151.624
C01446=1102.738,84.774,441.905,177.152,14.337,151.625
C01447=1102.732,84.524,441.923,177.149,14.337,151.625
C01448=1102.727,84.275,441.941,177.147,14.337,151.626
C01449=1102.721,84.026,441.957,177.143,14.337,151.627
C01450=1102.715,83.776,441.975,177.141,14.337,151.627
C01451=1102.709,83.527,441.993,177.137,14.337,151.628
C01452=1102.704,83.278,442.010,177.135,14.337,151.629
C01453=1102.698,83.029,442.028,177.132,14.338,151.629
C01454=1102.692,82.779,442.046,177.128,14.337,151.630
C01455=1102.686,82.530,442.063,177.126,14.338,151.631
C01456=1102.681,82.280,442.080,177.123,14.338,151.631
C01457=1102.675,82.031,442.098,177.120,14.338,151.632
C01458=1102.670,81.782,442.116,177.117,14.338,151.632
C01459=1102.664,81.532,442.133,177.115,14.338,151.633
C01460=1102.659,81.283,442.150,177.111,14.338,151.634
C01461=1102.653,81.033,442.168,177.109,14.338,151.634
C01462=1102.647,80.784,442.186,177.105,14.337,151.635
C01463=1102.642,80.535,442.203,177.103,14.338,151.636
C01464=1102.636,80.263,442.221,177.100,14.338,151.636
C01465=1102.629,79.990,442.241,177.096,14.338,151.637
C01466=1102.623,79.719,442.260,177.093,14.337,151.638
C01467=1102.617,79.446,442.278,177.090,14.338,151.638
C01468=1102.611,79.197,442.296,177.087,14.337,151.639
C01469=1102.605,78.948,442.314,177.085,14.337,151.640
C01470=1102.600,78.699,442.331,177.082,14.338,151.640
C01471=1102.595,78.449,442.348,177.078,14.337,151.641
C01472=1102.588,78.200,442.365,177.076,14.337,151.642
C01473=1102.582,77.950,442.383,177.073,14.337,151.642
C01474=1102.577,77.701,442.400,177.070,14.337,151.643
C01475=1102.572,77.452,442.417,177.067,14.337,151.644
C01476=1102.566,77.202,442.434,177.065,14.337,151.644
C01477=1102.560,76.953,442.451,177.061,14.337,151.645
C01478=1102.554,76.704,442.469,177.059,14.337,151.645
C01479=1102.549,76.454,442.486,177.056,14.338,151.646
C01480=1102.543,76.205,442.503,177.053,14.337,151.647
C01481=1102.537,75.956,442.520,177.050,14.337,151.647
C01482=1102.531,75.706,442.538,177.048,14.337,151.648
C01483=1102.526,75.457,442.555,177.044,14.337,151.649
C01484=1102.520,75.207,442.571,177.042,14.337,151.649
C01485=1102.514,74.958,442.589,177.038,14.337,151.650
C01486=1102.509,74.709,442.606,177.036,14.337,151.650
C01487=1102.503,74.460,442.623,177.033,14.337,151.651
C01488=1102.497,74.210,442.640,177.030,14.336,151.652
C01489=1102.491,73.961,442.658,177.027,14.337,151.652
C01490=1102.486,73.711,442.674,177.025,14.337,151.653
C01491=1102.480,73.462,442.691,177.021,14.336,151.654
C01492=1102.475,73.213,442.708,177.019,14.337,151.654
C01493=1102.469,72.964,442.725,177.016,14.337,151.655
C01494=1102.463,72.714,442.742,177.013,14.336,151.655
C01495=1102.457,72.464,442.760,177.011,14.336,151.656
C01496=1102.451,72.215,442.776,177.008,14.336,151.656
C01497=1102.446,71.966,442.794,177.005,14.336,151.657
C01498=1102.441,71.716,442.811,177.002,14.336,151.658
C01499=1102.435,71.467,442.827,177.000,14.336,151.658
C01500=1102.429,71.218,442.845,176.996,14.336,151.659
C01501=1102.423,70.969,442.861,176.994,14.336,151.660
C01502=1102.418,70.720,442.878,176.991,14.336,151.660
C01503=1102.412,70.470,442.895,176.988,14.336,151.661
C01504=1102.406,70.221,442.911,176.985,14.336,151.661
C01505=1102.401,69.972,442.929,176.983,14.336,151.662
C01506=1102.394,69.721,442.946,176.980,14.335,151.663
C01507=1102.389,69.472,442.963,176.977,14.335,151.663
C01508=1102.383,69.223,442.979,176.975,14.335,151.664
C01509=1102.378,68.973,442.996,176.971,14.335,151.664
C01510=1102.372,68.724,443.013,176.969,14.335,151.665
C01511=1102.366,68.475,443.030,176.966,14.335,151.665
C01512=1102.360,68.226,443.046,176.963,14.335,151.666
C01513=1102.355,67.976,443.063,176.960,14.335,151.667
C01514=1102.349,67.727,443.080,176.958,14.335,151.667
C01515=1102.344,67.478,443.097,176.955,14.334,151.668
C01516=1102.338,67.228,443.113,176.952,14.334,151.668
C01517=1102.332,66.979,443.130,176.950,14.334,151.669
C01518=1102.326,66.730,443.147,176.946,14.334,151.670
C01519=1102.321,66.480,443.164,176.944,14.334,151.670
C01520=1102.314,66.230,443.181,176.942,14.334,151.671
C01521=1102.309,65.981,443.197,176.938,14.333,151.671
C01522=1102.303,65.731,443.214,176.936,14.333,151.672
C01523=1102.298,65.482,443.231,176.933,14.333,151.672
C01524=1102.292,65.233,443.248,176.930,14.333,151.673
C01525=1102.286,64.983,443.264,176.928,14.333,151.674
C01526=1102.281,64.734,443.281,176.925,14.333,151.674
C01527=1102.275,64.484,443.297,176.922,14.332,151.675
C01528=1102.268,64.212,443.315,176.919,14.333,151.675
C01529=1102.262,63.940,443.333,176.916,14.332,151.676
C01530=1102.256,63.669,443.352,176.913,14.332,151.677
C01531=1102.249,63.397,443.369,176.910,14.332,151.677
C01532=1102.244,63.146,443.387,176.907,14.332,151.678
C01533=1102.238,62.897,443.403,176.905,14.332,151.678
C01534=1102.232,62.647,443.419,176.902,14.331,151.679
C01535=1102.226,62.398,443.435,176.899,14.331,151.680
C01536=1102.221,62.148,443.452,176.897,14.331,151.680
C01537=1102.215,61.899,443.469,176.894,14.331,151.681
C01538=1102.209,61.650,443.485,176.891,14.331,151.681
C01539=1102.203,61.400,443.501,176.889,14.331,151.682
C01540=1102.197,61.151,443.518,176.885,14.331,151.683
C01541=1102.192,60.901,443.534,176.883,14.330,151.683
C01542=1102.185,60.653,443.551,176.881,14.330,151.684
C01543=1102.179,60.403,443.567,176.878,14.330,151.684
C01544=1102.174,60.154,443.584,176.875,14.330,151.685
C01545=1102.168,59.904,443.601,176.872,14.330,151.685
C01546=1102.162,59.655,443.617,176.870,14.330,151.686
C01547=1102.156,59.406,443.633,176.867,14.329,151.686
C01548=1102.151,59.156,443.650,176.864,14.329,151.687
C01549=1102.146,58.907,443.666,176.862,14.329,151.688
C01550=1102.140,58.657,443.681,176.858,14.329,151.688
C01551=1102.134,58.408,443.698,176.856,14.329,151.689
C01552=1102.128,58.159,443.714,176.854,14.329,151.689
C01553=1102.123,57.909,443.731,176.850,14.328,151.690
C01554=1102.117,57.660,443.747,176.848,14.328,151.690
C01555=1102.111,57.410,443.763,176.846,14.328,151.691
C01556=1102.105,57.161,443.779,176.843,14.328,151.691
C01557=1102.099,56.912,443.796,176.840,14.327,151.692
C01558=1102.093,56.662,443.812,176.838,14.327,151.692
C01559=1102.088,56.413,443.829,176.835,14.327,151.693
C01560=1102.082,56.163,443.845,176.832,14.327,151.694
C01561=1102.076,55.913,443.861,176.829,14.327,151.694
C01562=1102.071,55.665,443.876,176.827,14.326,151.695
C01563=1102.065,55.415,443.893,176.824,14.326,151.695
C01564=1102.059,55.166,443.909,176.821,14.326,151.696
C01565=1102.053,54.917,443.925,176.819,14.326,151.696
C01566=1102.048,54.667,443.942,176.817,14.326,151.697
C01567=1102.042,54.417,443.958,176.814,14.325,151.697
C01568=1102.036,54.168,443.974,176.811,14.325,151.698
C01569=1102.030,53.918,443.990,176.809,14.325,151.698
C01570=1102.025,53.670,444.006,176.806,14.324,151.699
C01571=1102.019,53.420,444.022,176.803,14.324,151.699
C01572=1102.013,53.170,444.038,176.801,14.324,151.700
C01573=1102.007,52.921,444.054,176.799,14.324,151.700
C01574=1102.002,52.672,444.070,176.795,14.323,151.701
C01575=1101.996,52.422,444.087,176.793,14.323,151.701
C01576=1101.991,52.173,444.102,176.791,14.323,151.702
C01577=1101.985,51.923,444.119,176.788,14.322,151.702
C01578=1101.979,51.674,444.135,176.785,14.322,151.703
C01579=1101.974,51.424,444.150,176.783,14.322,151.704
C01580=1101.968,51.175,444.167,176.780,14.321,151.704
C01581=1101.962,50.926,444.183,176.777,14.322,151.705
C01582=1101.956,50.677,444.199,176.775,14.321,151.705
C01583=1101.951,50.427,444.214,176.772,14.321,151.706
C01584=1101.945,50.177,444.231,176.769,14.320,151.706
C01585=1101.939,49.928,444.247,176.767,14.321,151.707
C01586=1101.934,49.679,444.262,176.765,14.320,151.707
C01587=1101.928,49.429,444.278,176.762,14.320,151.708
C01588=1101.922,49.179,444.294,176.759,14.319,151.708
C01589=1101.916,48.930,444.310,176.757,14.319,151.709
C01590=1101.911,48.681,444.326,176.755,14.319,151.709
C01591=1101.905,48.431,444.342,176.751,14.319,151.710
C01592=1101.899,48.159,444.360,176.749,14.318,151.710
C01593=1101.893,47.887,444.377,176.746,14.318,151.711
C01594=1101.887,47.614,444.394,176.743,14.318,151.711
C01595=1101.881,47.341,444.411,176.740,14.317,151.712
C01596=1101.875,47.092,444.427,176.738,14.317,151.712
C01597=1101.869,46.843,444.443,176.736,14.317,151.713
C01598=1101.864,46.593,444.458,176.732,14.316,151.713
C01599=1101.858,46.344,444.475,176.730,14.316,151.714
C01600=1101.852,46.094,444.490,176.728,14.315,151.714
C01601=1101.847,45.845,444.506,176.725,14.316,151.715
C01602=1101.841,45.595,444.522,176.723,14.315,151.715
C01603=1101.835,45.346,444.538,176.720,14.315,151.716
C01604=1101.830,45.096,444.553,176.718,14.314,151.716
C01605=1101.824,44.847,444.569,176.716,14.314,151.717
C01606=1101.819,44.598,444.585,176.712,14.314,151.717
C01607=1101.813,44.348,444.600,176.710,14.313,151.718
C01608=1101.808,44.099,444.616,176.708,14.313,151.718
C01609=1101.802,43.849,444.632,176.705,14.312,151.719
C01610=1101.796,43.600,444.648,176.703,14.312,151.719
C01611=1101.791,43.350,444.663,176.700,14.312,151.720
C01612=1101.784,43.101,444.679,176.698,14.312,151.720
C01613=1101.779,42.851,444.694,176.695,14.311,151.721
C01614=1101.774,42.602,444.710,176.692,14.311,151.721
C01615=1101.768,42.353,444.726,176.690,14.311,151.722
C01616=1101.762,42.103,444.741,176.688,14.310,151.722
C01617=1101.756,41.854,444.756,176.685,14.310,151.723
C01618=1101.750,41.604,444.772,176.682,14.309,151.723
C01619=1101.745,41.354,444.788,176.680,14.309,151.724
C01620=1101.739,41.106,444.804,176.678,14.309,151.724
C01621=1101.734,40.856,444.819,176.675,14.308,151.725
C01622=1101.727,40.606,444.834,176.673,14.308,151.725
C01623=1101.722,40.358,444.850,176.670,14.308,151.726
C01624=1101.716,40.108,444.866,176.667,14.307,151.726
C01625=1101.711,39.858,444.881,176.665,14.307,151.726
C01626=1101.705,39.609,444.896,176.662,14.307,151.727
C01627=1101.699,39.359,444.912,176.660,14.306,151.727
C01628=1101.693,39.109,444.927,176.657,14.306,151.728
C01629=1101.688,38.860,444.943,176.655,14.305,151.728
C01630=1101.681,38.611,444.958,176.653,14.305,151.729
C01631=1101.676,38.361,444.974,176.650,14.305,151.729
C01632=1101.671,38.112,444.989,176.647,14.304,151.730
C01633=1101.665,37.862,445.005,176.645,14.304,151.730
C01634=1101.659,37.614,445.020,176.643,14.304,151.731
C01635=1101.653,37.364,445.035,176.641,14.303,151.731
C01636=1101.647,37.114,445.050,176.638,14.302,151.732
C01637=1101.642,36.865,445.065,176.635,14.303,151.732
C01638=1101.636,36.615,445.081,176.633,14.302,151.733
C01639=1101.630,36.366,445.097,176.631,14.302,151.733
C01640=1101.625,36.116,445.112,176.628,14.301,151.734
C01641=1101.618,35.867,445.127,176.625,14.301,151.734
C01642=1101.613,35.617,445.142,176.623,14.301,151.735
C01643=1101.607,35.367,445.158,176.621,14.300,151.735
C01644=1101.601,35.118,445.172,176.619,14.300,151.735
C01645=1101.596,34.869,445.188,176.615,14.300,151.736
C01646=1101.589,34.620,445.203,176.613,14.299,151.736
C01647=1101.584,34.370,445.218,176.611,14.299,151.737
C01648=1101.578,34.121,445.233,176.609,14.299,151.737
C01649=1101.572,33.871,445.249,176.606,14.298,151.738
C01650=1101.567,33.621,445.264,176.603,14.298,151.738
C01651=1101.561,33.372,445.279,176.601,14.297,151.739
C01652=1101.556,33.122,445.294,176.599,14.297,151.739
C01653=1101.549,32.873,445.309,176.596,14.296,151.740
C01654=1101.544,32.624,445.325,176.594,14.296,151.740
C01655=1101.538,32.374,445.340,176.592,14.295,151.740
C01656=1101.532,32.101,445.357,176.588,14.295,151.741
C01657=1101.526,31.829,445.373,176.586,14.295,151.742
C01658=1101.519,31.557,445.389,176.584,14.294,151.742
C01659=1101.513,31.284,445.406,176.581,14.294,151.743
C01660=1101.508,31.035,445.421,176.578,14.293,151.743
C01661=1101.501,30.786,445.436,176.576,14.293,151.743
C01662=1101.496,30.536,445.451,176.573,14.292,151.744
C01663=1101.490,30.287,445.466,176.571,14.292,151.744
C01664=1101.485,30.037,445.482,176.569,14.291,151.745
C01665=1101.478,29.788,445.496,176.567,14.291,151.745
C01666=1101.473,29.538,445.512,176.564,14.291,151.746
C01667=1101.467,29.288,445.526,176.561,14.290,151.746
C01668=1101.462,29.039,445.541,176.559,14.290,151.747
C01669=1101.456,28.789,445.556,176.557,14.290,151.747
C01670=1101.451,28.540,445.571,176.555,14.289,151.747
C01671=1101.444,28.290,445.586,176.552,14.289,151.748
C01672=1101.438,28.041,445.601,176.550,14.288,151.748
C01673=1101.433,27.791,445.616,176.547,14.288,151.749
C01674=1101.427,27.542,445.631,176.545,14.287,151.749
C01675=1101.422,27.292,445.646,176.543,14.287,151.750
C01676=1101.415,27.043,445.661,176.540,14.286,151.750
C01677=1101.409,26.794,445.676,176.538,14.286,151.750
C01678=1101.405,26.544,445.690,176.535,14.286,151.751
C01679=1101.398,26.294,445.705,176.533,14.286,151.751
C01680=1101.393,26.045,445.720,176.531,14.285,151.752
C01681=1101.387,25.795,445.735,176.528,14.284,151.752
C01682=1101.381,25.546,445.750,176.526,14.284,151.753
C01683=1101.375,25.297,445.765,176.524,14.284,151.753
C01684=1101.370,25.048,445.780,176.521,14.283,151.754
C01685=1101.364,24.797,445.794,176.519,14.283,151.754
C01686=1101.358,24.548,445.809,176.516,14.282,151.754
C01687=1101.352,24.298,445.824,176.514,14.282,151.755
C01688=1101.346,24.049,445.839,176.512,14.281,151.755
C01689=1101.340,23.800,445.854,176.510,14.281,151.756
C01690=1101.335,23.550,445.868,176.507,14.281,151.756
C01691=1101.329,23.300,445.883,176.504,14.280,151.757
C01692=1101.323,23.051,445.898,176.502,14.279,151.757
C01693=1101.317,22.802,445.913,176.500,14.279,151.757
C01694=1101.312,22.552,445.927,176.498,14.279,151.758
C01695=1101.306,22.303,445.942,176.496,14.278,151.758
C01696=1101.300,22.053,445.957,176.493,14.277,151.759
C01697=1101.294,21.803,445.971,176.491,14.277,151.759
C01698=1101.289,21.554,445.986,176.488,14.277,151.760
C01699=1101.283,21.305,446.001,176.486,14.276,151.760
C01700=1101.277,21.056,446.015,176.484,14.276,151.760
C01701=1101.271,20.805,446.030,176.481,14.275,151.761
C01702=1101.266,20.556,446.045,176.479,14.275,151.761
C01703=1101.260,20.307,446.059,176.477,14.274,151.762
C01704=1101.254,20.057,446.074,176.475,14.274,151.762
C01705=1101.248,19.808,446.088,176.473,14.273,151.762
C01706=1101.242,19.558,446.103,176.470,14.272,151.763
C01707=1101.237,19.308,446.118,176.467,14.272,151.763
C01708=1101.231,19.059,446.132,176.465,14.272,151.764
C01709=1101.225,18.809,446.146,176.463,14.272,151.764
C01710=1101.220,18.560,446.161,176.461,14.271,151.765
C01711=1101.213,18.310,446.176,176.459,14.271,151.765
C01712=1101.208,18.061,446.190,176.456,14.270,151.765
C01713=1101.203,17.812,446.205,176.454,14.270,151.766
C01714=1101.197,17.561,446.219,176.451,14.269,151.766
C01715=1101.191,17.312,446.234,176.449,14.269,151.767
C01716=1101.185,17.063,446.248,176.447,14.268,151.767
C01717=1101.179,16.813,446.263,176.445,14.268,151.767
C01718=1101.173,16.564,446.277,176.442,14.267,151.768
C01719=1101.168,16.315,446.291,176.440,14.267,151.768
C01720=1101.162,16.043,446.307,176.438,14.266,151.769
C01721=1101.155,15.772,446.323,176.435,14.265,151.769
C01722=1101.149,15.501,446.338,176.433,14.265,151.770
C01723=1101.142,15.230,446.354,176.430,14.265,151.770
C01724=1101.137,14.981,446.369,176.428,14.264,151.770
C01725=1101.131,14.731,446.383,176.425,14.263,151.771
C01726=1101.126,14.482,446.398,176.423,14.263,151.771
C01727=1101.120,14.232,446.412,176.421,14.263,151.772
C01728=1101.114,13.982,446.426,176.419,14.262,151.772
C01729=1101.108,13.733,446.440,176.417,14.262,151.772
C01730=1101.102,13.484,446.455,176.415,14.261,151.773
C01731=1101.096,13.234,446.469,176.412,14.260,151.773
C01732=1101.091,12.984,446.483,176.409,14.260,151.774
C01733=1101.085,12.735,446.498,176.407,14.260,151.774
C01734=1101.078,12.485,446.511,176.405,14.259,151.774
C01735=1101.073,12.236,446.526,176.403,14.259,151.775
C01736=1101.067,11.987,446.540,176.401,14.259,151.775
C01737=1101.061,11.737,446.555,176.398,14.257,151.776
C01738=1101.055,11.487,446.569,176.396,14.257,151.776
C01739=1101.050,11.238,446.582,176.394,14.257,151.776
C01740=1101.043,10.988,446.597,176.391,14.256,151.777
C01741=1101.038,10.738,446.611,176.389,14.256,151.777
C01742=1101.032,10.489,446.625,176.387,14.256,151.778
C01743=1101.027,10.240,446.640,176.385,14.255,151.778
C01744=1101.021,9.990,446.654,176.382,14.254,151.778
C01745=1101.015,9.740,446.668,176.380,14.254,151.779
C01746=1101.009,9.491,446.682,176.378,14.253,151.779
C01747=1101.002,9.241,446.696,176.376,14.253,151.780
C01748=1100.997,8.992,446.710,176.374,14.252,151.780
C01749=1100.991,8.743,446.724,176.372,14.252,151.780
C01750=1100.986,8.493,446.738,176.369,14.252,151.781
C01751=1100.980,8.243,446.752,176.366,14.251,151.781
C01752=1100.974,7.994,446.767,176.365,14.250,151.782
C01753=1100.968,7.744,446.781,176.362,14.249,151.782
C01754=1100.963,7.495,446.795,176.360,14.249,151.782
C01755=1100.956,7.245,446.808,176.358,14.249,151.783
C01756=1100.950,6.996,446.823,176.356,14.249,151.783
C01757=1100.945,6.746,446.837,176.354,14.248,151.783
C01758=1100.939,6.497,446.851,176.351,14.247,151.784
C01759=1100.933,6.246,446.865,176.349,14.246,151.784
C01760=1100.928,5.997,446.879,176.347,14.246,151.785
C01761=1100.921,5.748,446.893,176.345,14.245,151.785
C01762=1100.916,5.499,446.907,176.343,14.245,151.785
C01763=1100.910,5.249,446.921,176.340,14.245,151.786
C01764=1100.904,4.999,446.935,176.338,14.244,151.786
C01765=1100.899,4.749,446.949,176.336,14.244,151.787
C01766=1100.893,4.500,446.963,176.333,14.243,151.787
C01767=1100.887,4.251,446.976,176.331,14.242,151.787
C01768=1100.881,4.001,446.990,176.329,14.242,151.788
C01769=1100.876,3.752,447.004,176.327,14.241,151.788
C01770=1100.870,3.501,447.018,176.325,14.241,151.789
C01771=1100.864,3.252,447.032,176.323,14.240,151.789
C01772=1100.858,3.003,447.046,176.321,14.240,151.789
C01773=1100.853,2.753,447.059,176.319,14.240,151.790
C01774=1100.847,2.504,447.074,176.316,14.238,151.790
C01775=1100.841,2.255,447.088,176.314,14.238,151.790
C01776=1100.835,2.005,447.102,176.312,14.237,151.791
C01777=1100.829,1.755,447.115,176.310,14.237,151.791
C01778=1100.824,1.505,447.129,176.308,14.236,151.791
C01779=1100.818,1.256,447.143,176.305,14.236,151.792
C01780=1100.813,1.006,447.157,176.303,14.235,151.792
C01781=1100.806,0.757,447.170,176.301,14.235,151.793
C01782=1100.801,0.507,447.184,176.298,14.234,151.793
C01783=1100.795,0.258,447.198,176.296,14.233,151.793
C01784=1100.789,-0.011,447.213,176.294,14.233,151.794
C01785=1100.782,-0.281,447.227,176.292,14.233,151.794
C01786=1100.776,-0.549,447.242,176.289,14.232,151.795
C01787=1100.771,-0.819,447.258,176.287,14.231,151.795
C01788=1100.764,-1.068,447.271,176.285,14.231,151.795
C01789=1100.759,-1.317,447.285,176.283,14.230,151.796
C01790=1100.753,-1.567,447.299,176.281,14.229,151.796
C01791=1100.748,-1.817,447.313,176.279,14.229,151.796
C01792=1100.742,-2.066,447.326,176.277,14.228,151.797
C01793=1100.736,-2.316,447.340,176.275,14.228,151.797
C01794=1100.730,-2.566,447.354,176.272,14.227,151.797
C01795=1100.724,-2.816,447.367,176.270,14.226,151.798
C01796=1100.719,-3.065,447.380,176.268,14.226,151.798
C01797=1100.713,-3.315,447.394,176.266,14.225,151.799
C01798=1100.707,-3.564,447.408,176.264,14.225,151.799
C01799=1100.702,-3.814,447.421,176.262,14.224,151.799
C01800=1100.695,-4.063,447.435,176.260,14.224,151.800
C01801=1100.690,-4.312,447.449,176.257,14.223,151.800
C01802=1100.684,-4.562,447.462,176.256,14.223,151.800
C01803=1100.678,-4.811,447.476,176.253,14.222,151.801
C01804=1100.672,-5.062,447.490,176.250,14.221,151.801
